# B&R Automation Studio project Doctor
Automation Studio 4.9

## Configuration 5Drive

CPU 4PPC70.0702-20B, AutomationRuntime J4.93, Build 4.1.2, Vc V4.72.6

### Hardware
```
4PPC70_0702_20B : 4PPC70.0702-20B v1.5.4.0
  Connector IF2:
    ActivateDevice = 1
  ConfigurationID = TensionCtl_Config1
  FileDevice1
  FileDeviceName1 = USER
  FileDevicePath1 = USER_PATH
  KeyMappingFile = VC\4PPC70_0702_20B.dis
```

## Configuration Doctoring

CPU 4PPC70.0702-20B, AutomationRuntime J4.93, Build 4.1.2, Safety 0.0, Vc V4.73.3

### Task classes (Cpu.sw)
```
Cyclic#1 (cycle 2000 us, tolerance 4000 us):
  HS_Inp_Doc <- Doctoring.HS_Inp_Doct.prg
  EPLCom_Drv <- EPLCom.EPLCom_Drv1.prg
Cyclic#2 (cycle 10000 us):
  LS_Inp_OP <- Doctoring.LS_Inp_OP.prg
Cyclic#4:
  HMI <- HMI.prg
  Alarms <- Alarms.prg
  EPLCom_Dr1 <- EPLCom.EPLCom_Drv2.prg
DataObjects: Acp10sys
VcDataObjects: Vis <- Vis.dob
Binaries: udbdef, FWRules, TCData, vcctext, arialbd, vcpdi855, vcmgr, vcdsint, vcdsloc, vcbclass, vcfntttf, vctcal, vcshared, vcrt, vcpk, vccbmp, vcfile, vccbtn, vccslider, vccdt, vcptelo, vcalarm, vccnum, vcpdsw, arial, vccovl, vccalarm, vccstr, vcpdi815, vcpfppc7, vcgclass, vcpdihd, vcnet, Vis01, Vis03, vcpkat, Vis02, vcpdvnc, vccline, visvc, vclibvc, vcclbox, vccshape, acp10cfg, Acp10map, arconfig, User, iomap, asfw, ashwac, ashwd, sysconf, Role, vcpfar00, vcxml, vcchspot, vcchtml, vccurl, Vis_Re02, Vis_Re01, Vis_Re03, Vis_Re, vcctrend
Libraries: NcGlobal, sys_lib, brsystem, runtime, LoopConR, LoopCont, Acp10_MC, Acp10man, Acp10par, AsBrMath, Acp10sim, asstring, standard, vclib, visapi, AsEPL, Library, astime, fileio, powerlnk, asieccon, dataobj, vcresman
```

### Hardware
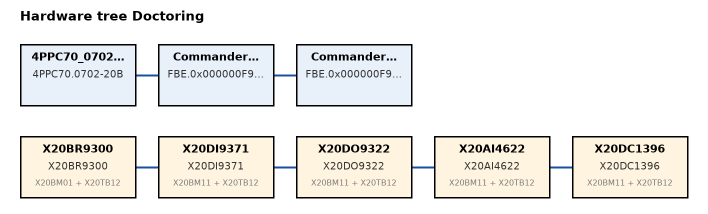
```
4PPC70_0702_20B : 4PPC70.0702-20B v1.5.4.0
  Connector IF1:
    CycleTime = 500
    MuxPrescaler = 2
  Connector IF2:
    ActivateDevice = 1
    Mode = Manual
    InternetAddress = 192.168.111.50
    SubnetMask = 255.255.255.0
    InaNodeNumber = 3
    Vnc1
    VncVcObjectName1 = Vis
    VncKeyMappingFile1 = VC\PS2-Keyboard.dis
    VncAuthentication1 = 1
    VncPasswordViewControl1 = v
    ActivateSnmp = 2
  Connector IF5:
    CycleTime = 1000
    BusLength = 500
  ConfigurationID = TensionCtl_Config1
  SimulationInaNodeNumber = 3
  PermanentPvSize = 5000
  RemanentGlobalPvSize = 10000
  EnableUsbRemoteInstall = 1
  EnableCfRemoteInstall = 1
  RebootReset = 2
  Connections = 8
  TimerDeviceType = EPLX2X
  TimerDevice = 4PPC70_0702_20B.IF1
  IdleTaskClass = 4
  TaskClassIdleTime = 4000
  Cyclic1Duration = 2000
  Cyclic1Tolerance = 4000
  Cyclic2Duration = 10000
  Cyclic5Duration = 500000
  Cyclic5Tolerance = 500000
  FileDevice1
  FileDeviceName1 = USER
  FileDevicePath1 = USER_PATH
  ActivateOpcUa = 1
  OpcUaInformationModels_PV_Version = 1
  VcObjectName = Vis
  KeyMappingFile = VC\4PPC70_0702_20B.dis
Commander_C200_RFC_UnWind : FBE.0x000000F9_Commander C200 RFC_A vV01.01.12.04 (OrderNumber=Commander C200 RFC_A)  [PLK1 -> 4PPC70_0702_20B.IF1 (NodeNumber=3) [Cable Type=PowerlinkCable, Length=10, Version=1.0.0.3]; PLK2 -> Commander_C200_RFC_Wind.PLK1 (NodeNumber=3) [Cable Type=PowerlinkCable, Length=10, Version=1.0.0.3]]
  DummyDeviceType = on
  p2001s05_direction = wo
  p2001s05_value = 5
  p2001s15_value = 0
  p2001s18_direction = wo
  p2004s01_direction = ro
  p2005s01_direction = ro
  p2005s03_direction = ro
  p2005s04_direction = ro
  p2007s01_direction = ro
  p200Es08_value = 0
  p200Es19_value = 0
  p2014s15_value = 
  p6040_value = 0
Commander_C200_RFC_Wind : FBE.0x000000F9_Commander C200 RFC_A vV01.01.12.04 (OrderNumber=Commander C200 RFC_A)  [PLK1 -> Commander_C200_RFC_UnWind.PLK2 (NodeNumber=4) [Cable Type=PowerlinkCable, Length=10, Version=1.0.0.3]]
  p2001s05_direction = wo
  p2001s18_direction = wo
  p2004s01_direction = ro
  p2005s01_direction = ro
  p2005s03_direction = ro
  p2005s04_direction = ro
X20AI4622 : X20AI4622 v1.5.0.0  [SS1 -> X20TB12g.SS; SL -> X20BM11f.SL1]
  Supervision = off
X20BM01 : X20BM01 v2.2.0.0
X20BM11b : X20BM11 v1.1.0.0  [X2X1 -> X20BM01.X2X2]
X20BM11d : X20BM11 v1.1.0.0  [X2X1 -> X20BM11b.X2X2]
X20BM11f : X20BM11 v1.1.0.0  [X2X1 -> X20BM11d.X2X2]
X20BM11h : X20BM11 v1.1.0.0  [X2X1 -> X20BM11f.X2X2]
X20BR9300 : X20BR9300 v1.3.0.0  [SS1 -> X20TB12.SS; SL -> X20BM01.SL1; X2X1 -> 4PPC70_0702_20B.IF5 [Cable Type=X2XCable, Length=10, Version=1.0.0.3]]
  Supervision = off
X20DC1396 : X20DC1396 v1.4.0.0  [SS1 -> X20TB12i.SS; SL -> X20BM11h.SL1]
  Supervision = off
X20DI9371 : X20DI9371 v1.6.0.0  [SS1 -> X20TB12c.SS; SL -> X20BM11b.SL1]
  Supervision = off
X20DO9322 : X20DO9322 v1.6.0.0  [SS1 -> X20TB12e.SS; SL -> X20BM11d.SL1]
  Supervision = off
  StatusInfo = off
X20TB12 : X20TB12 v1.0.0.0
X20TB12c : X20TB12 v1.0.0.0
X20TB12e : X20TB12 v1.0.0.0
X20TB12g : X20TB12 v1.0.0.0
X20TB12i : X20TB12 v1.0.0.0
```

### Cpu.per - 4PPC70_0702_20B/Cpu.per
```iecst
VAR_CONFIG
	Wind AT %M0; (* *)
	UnWind AT %M220; (* *)
	Idler AT %M440; (* *)
END_VAR
```

### IoMap.iom - 4PPC70_0702_20B/IoMap.iom
```iecst
VAR_CONFIG
	Cyclic#1.::AI1[0] AT %IW."X20AI4622".AnalogInput01;
	Cyclic#1.::AI1[1] AT %IW."X20AI4622".AnalogInput02;
	Cyclic#1.::AI1[2] AT %IW."X20AI4622".AnalogInput03;
	Cyclic#1.::AI1[3] AT %IW."X20AI4622".AnalogInput04;
	::Enc_Value AT %IW."X20DC1396".Encoder01;
	::Drive_RW[0].Read_INT[0] AT %IW."Commander_C200_RFC_UnWind".Parameter40_StatusWord_I200A_S28;
	::Drive_RW[0].Write_UINT[0] AT %QW."Commander_C200_RFC_UnWind".Parameter5_JogReference_I2001_S05Out;
	Cyclic#2.::DI1[0] AT %IX."X20DI9371".DigitalInput01;
	Cyclic#2.::DI1[1] AT %IX."X20DI9371".DigitalInput02;
	Cyclic#2.::DI1[2] AT %IX."X20DI9371".DigitalInput03;
	Cyclic#2.::DI1[3] AT %IX."X20DI9371".DigitalInput04;
	Cyclic#2.::DI1[4] AT %IX."X20DI9371".DigitalInput05;
	Cyclic#2.::DI1[5] AT %IX."X20DI9371".DigitalInput06;
	Cyclic#2.::DI1[6] AT %IX."X20DI9371".DigitalInput07;
	Cyclic#2.::DI1[7] AT %IX."X20DI9371".DigitalInput08;
	Cyclic#2.::DI1[8] AT %IX."X20DI9371".DigitalInput09;
	Cyclic#2.::DI1[9] AT %IX."X20DI9371".DigitalInput10;
	Cyclic#2.::DI1[10] AT %IX."X20DI9371".DigitalInput11;
	Cyclic#2.::DI1[11] AT %IX."X20DI9371".DigitalInput12;
	Cyclic#2.::DO1[0] AT %QX."X20DO9322".DigitalOutput01;
	Cyclic#2.::DO1[1] AT %QX."X20DO9322".DigitalOutput02;
	Cyclic#2.::DO1[2] AT %QX."X20DO9322".DigitalOutput03;
	Cyclic#2.::DO1[3] AT %QX."X20DO9322".DigitalOutput04;
	Cyclic#2.::DO1[4] AT %QX."X20DO9322".DigitalOutput05;
	Cyclic#2.::DO1[5] AT %QX."X20DO9322".DigitalOutput06;
	Cyclic#2.::DO1[6] AT %QX."X20DO9322".DigitalOutput07;
	Cyclic#2.::DO1[7] AT %QX."X20DO9322".DigitalOutput08;
	Cyclic#2.::DO1[8] AT %QX."X20DO9322".DigitalOutput09;
	Cyclic#2.::DO1[9] AT %QX."X20DO9322".DigitalOutput10;
	Cyclic#2.::DO1[10] AT %QX."X20DO9322".DigitalOutput11;
	Cyclic#2.::DO1[11] AT %QX."X20DO9322".DigitalOutput12;
	::Drive_RW[0].Read_DINT[1] AT %ID."Commander_C200_RFC_UnWind".Parameter69_ReferenceInRpm_I2001_S45;
	::Drive_RW[0].Read_DINT[2] AT %ID."Commander_C200_RFC_UnWind".Parameter1_OutputFrequency_I2005_S01;
	::Drive_RW[0].Write_UINT[1] AT %QW."Commander_C200_RFC_UnWind".ControlWord_U16_I6040;
	::Drive_RW[0].Read_DINT[0] AT %ID."Commander_C200_RFC_UnWind".Parameter1_CurrentMagnitude_I2004_S01;
	::Drive_RW[0].Read_DINT[1] AT %ID."Commander_C200_RFC_UnWind".Parameter4_MotorRpm_I2005_S04;
	::Drive_RW[0].Read_DINT[3] AT %ID."Commander_C200_RFC_UnWind".Parameter3_OutputPower_I2005_S03;
	::Drive_RW[0].Write_DINT[0] AT %QD."Commander_C200_RFC_UnWind".Parameter22_PresetReference2_I2001_S16Out;
	::Drive_RW[1].Write_UINT[0] AT %QW."Commander_C200_RFC_Wind".Parameter5_JogReference_I2001_S05Out;
	::Drive_RW[1].Write_DINT[0] AT %QD."Commander_C200_RFC_Wind".Parameter22_PresetReference2_I2001_S16Out;
	::Drive_RW[1].Read_DINT[0] AT %ID."Commander_C200_RFC_Wind".Parameter1_CurrentMagnitude_I2004_S01;
	::Drive_RW[1].Read_DINT[2] AT %ID."Commander_C200_RFC_Wind".Parameter1_OutputFrequency_I2005_S01;
	::Drive_RW[1].Read_DINT[3] AT %ID."Commander_C200_RFC_Wind".Parameter3_OutputPower_I2005_S03;
	::Drive_RW[1].Read_DINT[1] AT %ID."Commander_C200_RFC_Wind".Parameter4_MotorRpm_I2005_S04;
	::Drive_RW[0].Read_INT[0] AT %IW."Commander_C200_RFC_UnWind".Parameter1_AnalogueInput1_I2007_S01;
	::Drive_RW[0].Write_DINT[0] AT %QD."Commander_C200_RFC_UnWind".Parameter21_PresetReference1_I2001_S15Out;
	::Drive_RW[0].Write_DINT[0] AT %QD."Commander_C200_RFC_UnWind".Parameter24_PresetReference4_I2001_S18Out;
	::Drive_RW[1].Write_DINT[0] AT %QD."Commander_C200_RFC_Wind".Parameter24_PresetReference4_I2001_S18Out;
END_VAR
```

## Configuration WndCLTensCtrl

### Acp10map.ncm - X20CP1586/Motion/Acp10map.ncm
```
NcMapping (NcSwId=Acp10, DisabledNodesAreHidden=False)
  NcObject gWinderAx (ModuleId=8V1022.001-2, Type=ncAXIS, Channel=1, AcoposSimulation=Complete, InitParameter=gWinderAxi, AcoposParameter=gWinderAxa, Disabled=FALSE, ModuleDisabled=FALSE)  // simulated winder axis
  NcObject gLineAx (ModuleId=8V1022.001-2, Type=ncV_AXIS, Channel=1, InitParameter=gLineAxi, AcoposParameter=gLineAxa, Disabled=FALSE, ModuleDisabled=FALSE)  // virtual master axis
```

## Configuration WndDcrCtrl

### Hardware
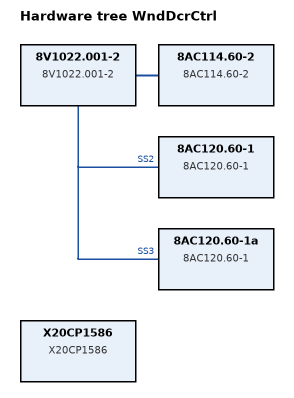
```
8AC114.60-2 : 8AC114.60-2 v1.0.0.8  [SS -> 8V1022.001-2.SS1; PLK1 -> X20CP1586.IF3 (NodeNumber=1) [Cable Type=PowerlinkCable, Length=10, Version=1.0.0.3]]
8AC120.60-1 : 8AC120.60-1 v2.2.0.0  [SS -> 8V1022.001-2.SS2]
8AC120.60-1a : 8AC120.60-1 v2.2.0.0  [SS -> 8V1022.001-2.SS3]
8V1022.001-2 : 8V1022.001-2 v2.2.0.0
  Simulate = complete
  ActiveMotorSimulation_r1 = on
  BothEndSwitchesAreNormallyOpen_r1 = on
  QuickStopIsNormallyOpen_r1 = on
X20CP1586 : X20CP1586 v1.10.0.0
  Connector IF1:
    ActivateIna = 0
  Connector IF2:
    ActivateDevice = 1
    EthInterfaceRedundant = 0
    InaPort = 11160
    Vnc1
    VncVcObjectName1 = Visu
    VncKeyMappingFile1 = VC\PS2-Keyboard.dis
    VncAuthentication1 = 1
    VncPasswordViewOnly1 = v
    VncPasswordViewControl1 = c
  Connector IF3:
    DNAConfiguration = manual
  ConfigurationID = DancerControl_Simulation
  Simulation = 1
  TimerDeviceType = SWIOTIMER
  SystemTick = 400
  TaskClassIdleTime = 400
  Cyclic1Duration = 400
  Cyclic1Tolerance = 0
  Cyclic2Duration = 800
  Cyclic2Tolerance = 0
  Cyclic3Duration = 10000
  Cyclic3Tolerance = 0
  Cyclic4Duration = 100000
  Cyclic4Tolerance = 100000
  Cyclic5Duration = 200000
  Cyclic5Tolerance = 200000
  Cyclic6Duration = 500000
  Cyclic6Tolerance = 500000
  Cyclic7Duration = 1000000
  Cyclic7Tolerance = 1000000
  Cyclic8Duration = 10000
  Cyclic8Tolerance = 30000000
```

### Acp10cfg.ncc - X20CP1586/Motion/Acp10cfg.ncc
```
NcConfiguration (Version=2.48.1, NcSwId=Acp10)
  ACP10CF1_typ:
    cnt_nettrc_rec_drive = 1500
    bufsize_trace_upload = 1200
    tc_nc_man_task = Cyclic #1
    glob_pv_as_ncobject = Yes
    ncsys_dl_broadcast = Yes
    ncsys_dl_acp_reset = Yes
    safemc_log_err_to_ax = Yes
    network_init:
      ncsw_init_execute = Yes
      automatic_execute = No
      node_nr_warning = Yes
      net_err_before_ncact = Yes
    nettrc:
      enter_parsecrec = Yes
      enter_ncaction = Yes
      save_ring_startidx = Yes
    cam_prof_download:
      cam_dat_dl_parallel = No
      tc_cam_dl_parallel = Task class for NC Manager task
    plk_if[0]:
      if_name = SL1.IF2
      tc_CycDat_PLCopen = Task class for NC Manager task
      mc_broadcast_extdat = No
    plk_if[1]:
      if_name = IF3
      tc_CycDat_PLCopen = Task class for NC Manager task
      mc_broadcast_extdat = No
```

### PvMap.vvm - X20CP1586/PvMap.vvm
```iecst
(*Simulation model input parameters*)
VAR_CONFIG
	Cyclic#3.::gControl.Winder.Power AT %Q.::SimModel:SimulationModel.Enable; (*Enable simulation modell if machine is ready*)
	Cyclic#3.::gControl.Line.SetVelocity AT %Q.::SimModel:SetLineVelocity; (*Connect control structure with simulation model*)
	Cyclic#3.::gControl.Winder.SetVelocity AT %Q.::SimModel:SetWinderVelocity; (*Connect control structure with simulation model*)
	Cyclic#3.::gControl.Winder.VelocityCorrection AT %Q.::SimModel:WinderVelocityCorrection; (*Connect control structure with simulation model*)
	Cyclic#3.::gControl.Winder.SetMotorTorque AT %Q.::SimModel:SetMotorTorque; (*Connect control structure with simulation model*)
	Cyclic#3.::gControl.Winder.InitSpeedController AT %Q.::SimModel:InitSpeedController; (*Connect control structure with simulation model*)
	Cyclic#3.::gControl.Winder.ActProportionalGain AT %Q.::SimModel:ActProportionalGain; (*Connect control structure with simulation model*)
	Cyclic#3.::gControl.Winder.ActIntegrationTime AT %Q.::SimModel:ActIntegrationTime; (*Connect control structure with simulation model*)
END_VAR
(*Simulation model output parameters*)
VAR_CONFIG
	::SimModel:SimulationModel.ActLinePosition AT %Q.Cyclic#2.::gControl.Line.ActPosition; (*Connect simulation model with control structure*)
	::SimModel:SimulationModel.ActWinderPosition AT %Q.Cyclic#2.::gControl.Winder.ActPosition; (*Connect simulation model with control structure*)
	::SimModel:SimulationModel.ActDancerPosition AT %Q.Cyclic#2.::gControl.ActDancerPosition; (*Connect simulation model with control structure*)
	::SimModel:SimulationModel.ActLineVelocity AT %Q.Cyclic#2.::gControl.Line.ActVelocity; (*Connect simulation model with control structure*)
	::SimModel:SimulationModel.ActWinderVelocity AT %Q.Cyclic#2.::gControl.Winder.ActVelocity; (*Connect simulation model with control structure*)
	::SimModel:SimulationModel.ActMotorTorque AT %Q.Cyclic#2.::gControl.Winder.ActMotorTorque; (*Connect simulation model with control structure*)
END_VAR
```

## Logical view

Binary libraries used (declarations not repeated): Acp10_MC 3.13.1, vclib

### Global.typ - Global data types
```iecst
TYPE
	ActVal_typ : 	STRUCT
		Input_Val : INT;
		Output_Val : INT;
		Scale : Scale_typ;
	END_STRUCT;
	Ax_GeneralRef : 	STRUCT
		MPM : MPM_Scale;
		RPM : RPM_Scale;
		PulsesPerRev : INT;
		MotorRating : MotorRating_typ;
	END_STRUCT;
	Ax_NonTensionCtl : 	STRUCT
		MPM : MPM_typ;
		Enable : BOOL;
		RPM : RPM_typ;
		Drive : Drive_typ;
		Dia : Diameter_Scale;
		StartingDia : UINT;
		MotorRating : MotorRating_typ;
	END_STRUCT;
	Ax_TensionCtl : 	STRUCT
		Tension : Tension_typ;
		MPM : MPM_typ;
		Enable : BOOL;
		RPM : RPM_typ;
		Drive : Drive_typ;
		Dia : Diameter_Scale;
		StartingDia : UINT;
		MotorRating : MotorRating_typ;
	END_STRUCT;
	Diameter_Scale : 	STRUCT
		InpMPM : INT;
		InpRPM : INT;
		ActDia : INT;
		MinDia : INT;
		MaxDia : INT;
	END_STRUCT;
	DigInp_typ : 	STRUCT
		Emergency_OK : BOOL;
		Jog_mode : BOOL;
		Production_mode : BOOL;
		MPM_Increase : BOOL;
		MPM_Decrease : BOOL;
		Safety_Trip : BOOL;
		Spare1 : BOOL;
		Spare2 : BOOL;
		Spare3 : BOOL;
		Spare4 : BOOL;
		Spare5 : BOOL;
		Spare6 : BOOL;
		Spare7 : BOOL;
		Spare8 : BOOL;
		Spare9 : BOOL;
		Spare10 : BOOL;
	END_STRUCT;
	DigOp_typ : 	STRUCT
		DriveOK : ARRAY[0..6]OF BOOL;
		Production_Enable : BOOL;
		Alarm_Lamp : BOOL;
		Safety_Trip : BOOL;
		Spare1 : BOOL;
		Spare2 : BOOL;
		Spare3 : BOOL;
		Spare4 : BOOL;
		Spare5 : BOOL;
		Spare6 : BOOL;
		Spare7 : BOOL;
		Spare8 : BOOL;
		Spare9 : BOOL;
		Spare10 : BOOL;
	END_STRUCT;
	Drive_typ : 	STRUCT
		Freq_Scal : Scale_typ;
		RPM_Scal : Scale_typ;
		Trq_Scal : Scale_typ;
		Current_Scal : Scale_typ;
		ActFreq : INT;
		Status : USINT;
		ActualTrq : INT;
		ActualAmp : INT;
		ActRPM : INT;
		Fault : USINT;
		Drive_Healthy : BOOL;
		Drive_Enable : BOOL;
	END_STRUCT;
	MPM_Scale : 	STRUCT
		InpDia : INT;
		InpRPM : INT;
		ActMPM : INT;
	END_STRUCT;
	MPM_typ : 	STRUCT
		SetMPM : INT;
		ActualMPM : INT;
		Enable : BOOL;
		Set : SetVal_typ;
		Actual : ActVal_typ;
	END_STRUCT;
	PIDPara_typ : 	STRUCT
		Y_max : INT;
		Y_min : INT;
		dY_max : REAL;
		Kp_sta : REAL;
		Tn_sta : REAL;
		Tv_sta : REAL;
		Tf_sta : REAL;
		WindDamp : REAL;
		Fbk_mode : REAL;
		d_mode : USINT;
		calc_mode : USINT;
		Attenu_val : REAL;
		Update : BOOL;
		Kp_mov : USINT;
		Tn_mov : USINT;
		Tv_mov : USINT;
		Tf_mov : USINT;
	END_STRUCT;
	RPM_Scale : 	STRUCT
		InpMPM : INT;
		InpDia : INT;
		ActRPM : INT;
		InpBits : INT;
	END_STRUCT;
	RPM_typ : 	STRUCT
		SetRPM : INT;
		ActualRPM : INT;
		Enable : BOOL;
		Set : SetVal_typ;
		Actual : ActVal_typ;
		PulsesPerRev : INT;
		GearRatio : USINT;
	END_STRUCT;
	Scale_typ : 	STRUCT
		InMin : INT;
		InMax : INT;
		OutMin : INT;
		OutMax : INT;
		Filter_tim : INT;
	END_STRUCT;
	SetVal_typ : 	STRUCT
		Output_Val : INT;
		Input_Val : INT;
		Scale : Scale_typ;
	END_STRUCT;
	Tension_typ : 	STRUCT
		Actual : ActVal_typ;
		Set : SetVal_typ;
		Enable : BOOL;
		SetTension : INT;
		ActualTension : INT;
		PID : PID_typ;
	END_STRUCT;
	DriveRW_typ : 	STRUCT
		Read_BOOL : ARRAY[0..9]OF BOOL;
		Read_UINT : ARRAY[0..9]OF UINT;
		Read_INT : ARRAY[0..9]OF INT;
		Read_USINT : ARRAY[0..9]OF USINT;
		Read_DINT : ARRAY[0..9]OF DINT;
		Read_UDINT : ARRAY[0..9]OF UDINT;
		Write_BOOL : ARRAY[0..9]OF BOOL;
		Write_INT : ARRAY[0..9]OF INT;
		Write_UINT : ARRAY[0..9]OF UINT;
		Write_USINT : ARRAY[0..9]OF USINT;
		Write_DINT : ARRAY[0..9]OF DINT;
		Write_UDINT : ARRAY[0..9]OF UDINT;
	END_STRUCT;
	MotorRating_typ : 	STRUCT
		RatedFreq : DINT;
		RatedCurrent : DINT;
		RatedSpeed : DINT;
		RatedVoltage : INT;
		RatedPF : INT;
	END_STRUCT;
	PID_typ : 	STRUCT
		Prop_Gain : INT;
		Intg_Gain : INT;
		Derv_Gain : INT;
		UpperLimit : INT;
		LowerLimit : INT;
		Enable : USINT;
		Reference_Add : INT;
		Feedback_Add : INT;
		Output : INT;
		Error : INT;
	END_STRUCT;
END_TYPE
```

### Global.var - Global variables
```iecst
VAR
	AI1 : ARRAY[0..4] OF INT;
	AI2 : ARRAY[0..3] OF INT;
	AI3 : ARRAY[0..4] OF INT;
	Alarm : ARRAY[0..99] OF BOOL;
	Alarm_cnt : USINT;
	Alarm_mc : ARRAY[0..99] OF BOOL;
	Alarm_new : BOOL;
	AO1 : ARRAY[0..3] OF INT;
	Axis_Motor : INT;
	Backbtn : INT;
	CurrPage : USINT;
	DataRead_INT : {REDUND_UNREPLICABLE} INT := 0;
	DataRead_UINT : UINT;
	DataTobeRead_INT : INT;
	DataTobeSent_UINT : UINT;
	DI1 : ARRAY[0..11] OF BOOL;
	DI2 : ARRAY[0..11] OF BOOL;
	DigInp : DigInp_typ;
	DigOp : DigOp_typ;
	DO1 : ARRAY[0..11] OF BOOL;
	DO2 : ARRAY[0..11] OF BOOL;
	Drive_RW : ARRAY[0..4] OF DriveRW_typ;
	DrvComm : BOOL;
	Enc_Value : INT;
	error : UINT;
END_VAR
VAR RETAIN
	Idler : Ax_GeneralRef;
END_VAR
VAR
	InFeed : Ax_TensionCtl;
END_VAR
VAR CONSTANT
	INFEED : USINT := 1;
END_VAR
VAR
	LastPage : USINT;
	LoginSuccessful : BOOL;
END_VAR
VAR CONSTANT
	MAIN : USINT := 4;
END_VAR
VAR
	MainDrive : Ax_NonTensionCtl;
END_VAR
VAR CONSTANT
	MAX_AXES : USINT := 5;
END_VAR
VAR
	NewPage : USINT;
	NewPageReq : USINT;
	OutFeed : Ax_TensionCtl;
END_VAR
VAR CONSTANT
	OUTFEED : USINT := 2;
END_VAR
VAR
	PageCall : BOOL;
	ParamChange : BOOL;
END_VAR
VAR CONSTANT
	PLC_INTF : STRING[20] := 'IF1';
END_VAR
VAR
	PrevPage : USINT;
	PrevPageTemp : USINT;
END_VAR
VAR CONSTANT
	PulsesPerRev : INT := 0;
END_VAR
VAR
	PulsesPerSec : INT;
	SavePID : BOOL;
	Save : BOOL;
	Statusdp_alarm : UINT;
	Statusdp_blink : UINT;
	status_gettime : UINT;
	TempPropGain : INT;
	TempIntgGain : INT;
	TempDervGain : INT;
	TempPIDFeedback : INT;
	TempPIDRef : INT;
	TempCurrent : DINT;
	TempFreq : DINT;
	TempPF : INT;
	TempSpeed : DINT;
	TempVoltage : INT;
END_VAR
VAR RETAIN
	UnWind : Ax_TensionCtl;
END_VAR
VAR CONSTANT
	UNWINDER : USINT := 0;
END_VAR
VAR
	UnWindpara : LCPIDpara;
	UserAccessLevel : USINT;
END_VAR
VAR RETAIN
	Wind : Ax_TensionCtl;
END_VAR
VAR CONSTANT
	WINDER : USINT := 3;
END_VAR
VAR
	Tune_Enable : BOOL;
	Axis_MotorTune : USINT;
END_VAR
```


### Program Logical/UnWindTC (IEC)

#### Cyclic.st
```iecst
PROGRAM _CYCLIC
	(* Insert code here *)
	(* PID parameters *)
	LCPIDpara_0.enable := start;
	LCPIDpara_0.enter  := paraEnter;
	LCPIDpara_0();		(* LCPIDpara function block call *)
	paraEnter := 0;

	(* PID controller *)
	LCPID_0.enable   := start;
	LCPID_0.ident    := LCPIDpara_0.ident; (* ident of PIDpara -> provides parameters (Kp, Tn, Tv, ...) *)
	LCPID_0.W        := setValue;
	LCPID_0.X        := actValue;
	LCPID_0.basetime := baseLCCounter.mscnt;
	LCPID_0();		(* LCPID function block call *)
	manipulatedVar := LCPID_0.Y;

END_PROGRAM
```

#### Init.st
```iecst
PROGRAM _INIT
	(* Insert code here *)
	(* Parameters for PID controller *)
	UnWindPID.A        := 0;
	UnWindPID.Y_man    := 0;
	UnWindPID.Y_fbk    := 0;
	UnWindPID.hold_I   := FALSE;
	UnWindPID.out_mode := LCPID_OUT_MODE_AUTO;

	(* Parameters for PID controller *)
	LCPID_0.A        := 0;
	LCPID_0.Y_man    := 0;
	LCPID_0.Y_fbk    := 0;
	LCPID_0.hold_I   := FALSE;
	LCPID_0.out_mode := LCPID_OUT_MODE_AUTO;

	(* Parameters for PT2 element *)
	LCRPT2_0.V     := 0.039;
	LCRPT2_0.T1    := 0.9;
	LCRPT2_0.T2    := 15.3;
	LCRPT2_0.y_set := 0.0;
	LCRPT2_0.set   := 0;

END_PROGRAM
```

### Program Logical/HMI (IEC)

#### Variables.var
```iecst
VAR
	CheckCredentials : BOOL;
	ErrorMessage : STRING[80];
	i : INT;
	Init : BOOL;
	InputPassword : STRING[80]; (*Input taken from HMI*)
	InputUsername : STRING[80]; (*Input taken from HMI*)
	CurrentYear : UINT;
	CurrentSecond : USINT;
	CurrentMonth : USINT;
	CurrentMinute : USINT;
	CurrentHour : USINT;
	CurrentDay : USINT;
	NewYear : UINT;
	NewSecond : USINT;
	NewMonth : USINT;
	NewMinute : USINT;
	NewHour : USINT;
	NewDay : USINT;
	DateTimeSet : UINT; (*Confirms if new date/time was set successfully*)
	SetNewDateTime : BOOL; (*Trigger to apply new date/time*)
	RTC_Get : RTCtime_typ; (*Structure to read current date and time*)
	RTC_Set : RTCtime_typ; (*Structure to set current date and time*)
	Status_RTC : UINT;
	temp_var : BOOL;
	startdly : BOOL;
	dlycnt : USINT;
	WelcomeTimer : TON_10ms;
END_VAR
```

#### Cyclic.st
```iecst
PROGRAM _CYCLIC
	// Time
	// Reads current date/time from PLC's RTC

	RTC_gettime(ADR(RTC_Get));  // Call PLC's built-in RTC function

	// Update outputs for display
	CurrentYear   := RTC_Get.year;
	CurrentMonth  := RTC_Get.month;
	CurrentDay    := RTC_Get.day;
	CurrentHour   := RTC_Get.hour;
	CurrentMinute := RTC_Get.minute;
	CurrentSecond := RTC_Get.second;

	// Set Date and Time when 'Set Date Time' button is pressed
	IF SetNewDateTime THEN
		IF(temp_var = 0)THEN
			Status_RTC	:= 1;
			temp_var	:= 1;
		END_IF

		RTC_Set.year    := NewYear;
		RTC_Set.month   := NewMonth;
		RTC_Set.day     := NewDay;
		RTC_Set.hour    := NewHour;
		RTC_Set.minute  := NewMinute;
		RTC_Set.second  := NewSecond;

		// Call RTC set function
		Status_RTC := RTC_settime(ADR(RTC_Set));  // Returns TRUE if successful

		IF(Status_RTC = 0)THEN
			SetNewDateTime	:= 0;
			temp_var		:= 0;
		END_IF

	END_IF;

	// Login check
	//IF(CurrPage > 0 AND CurrPage < 13) THEN
	IF (InputUsername = 'Admin' AND InputPassword = '1234') THEN
		LoginSuccessful := TRUE;
		UserAccessLevel := 1;	// Full access
		CheckCredentials := TRUE;
		ErrorMessage := 'Logged in';
	ELSE
		LoginSuccessful := FALSE;
		UserAccessLevel := 0;	// No input access
		CheckCredentials := FALSE;
		ErrorMessage := 'Wrong user name or password';
	END_IF;

	ErrorMessage := '';   	// Clear any previous message
	InputUsername := '';	// Clear InputUsername field
	InputPassword := '';	// Clear InputPassword field
	//END_IF

	IF(Alarm_new = 1)THEN
		Statusdp_alarm	:= 0;
	ELSE
		Statusdp_alarm	:= 1;
	END_IF

	IF((NewPageReq <> CurrPage) AND (dlycnt = 0)) THEN
		PrevPage := CurrPage;
		NewPage := NewPageReq;
		startdly	:= 0;
	END_IF

	IF(Backbtn = 1) THEN
		PrevPageTemp 	:= PrevPage;
		PrevPage 		:= CurrPage;
		NewPage 		:= PrevPageTemp;
		startdly		:= 1;
		Backbtn 		:= 0;
	END_IF

	IF((CurrPage = 0)AND (NewPageReq = 0))THEN
		WelcomeTimer.IN	:= 1;
		WelcomeTimer.PT	:= 500;
		IF(WelcomeTimer.Q = 1)THEN
			NewPageReq		:= 1;
			WelcomeTimer.IN	:= 0;
		END_IF
	END_IF

	WelcomeTimer();

	IF(startdly = 1)THEN
		dlycnt 		:= dlycnt + 1;
		NewPageReq 	:= CurrPage;
		IF(dlycnt = 3)THEN
			startdly	:= 0;
			dlycnt		:= 0;
		END_IF
	END_IF

END_PROGRAM
```

#### Init.st
```iecst
PROGRAM _INIT
		(*Input of Tension Sensor for 4 axes except main drive *)
	AI1[0]	:= 0;	(*Unwinder Loadcell *)
	AI1[1]	:= 0;	(* Infeed Loadcell *)
	AI1[2]	:= 0;	(* Outfeed Loadcell *)
	AI1[3]	:= 0;	(* Winder Load cell *)
	AI1[4]	:= 0;	(* Dummy Load cell for Main Drive *)

	AI2[0]	:= 0;
	AI2[1]	:= 0;
	AI2[2]	:= 0;
	AI2[3]	:= 0; (*This input is configured for MAIN RPM calculation *)

	(* Input for RPM measurement from drive AI for 4 axes except Winder RPM*)
	AI3[0]	:= 0;   (* Unwinder RPM *)
	AI3[1]	:= 0;	(* Infeed RPM *)
	AI3[2]	:= 0;	(* Outfeed RPM *)
	AI3[3]	:= 0;	(* Winder RPM *)
	AI3[4]	:= 0;	(*This input is configured from AI2[3] for MAIN RPM *)

	AO1[0]	:= 0;
	AO1[1]	:= 0;
	AO1[2]	:= 0;
	AO1[3]	:= 0;

	DI1[0]	:= 0;
	DI1[1]	:= 0;
	DI1[2]	:= 0;
	DI1[3]	:= 0;
	DI1[4]	:= 0;
	DI1[5]	:= 0;
	DI1[6]	:= 0;
	DI1[7]	:= 0;
	DI1[8]	:= 0;
	DI1[9]	:= 0;
	DI1[10]	:= 0;
	DI1[11]	:= 0;

	DI2[0]	:= 0;
	DI2[1]	:= 0;
	DI2[2]	:= 0;
	DI2[3]	:= 0;
	DI2[4]	:= 0;
	DI2[5]	:= 0;
	DI2[6]	:= 0;
	DI2[7]	:= 0;
	DI2[8]	:= 0;
	DI2[9]	:= 0;
	DI2[10]	:= 0;
	DI2[11]	:= 0;

	DO1[0]	:= 0;
	DO1[1]	:= 0;
	DO1[2]	:= 0;
	DO1[3]	:= 0;
	DO1[4]	:= 0;
	DO1[5]	:= 0;
	DO1[6]	:= 0;
	DO1[7]	:= 0;
	DO1[8]	:= 0;
	DO1[9]	:= 0;
	DO1[10]	:= 0;
	DO1[11]	:= 0;

	DO2[0]	:= 0;
	DO2[1]	:= 0;
	DO2[2]	:= 0;
	DO2[3]	:= 0;
	DO2[4]	:= 0;
	DO2[5]	:= 0;
	DO2[6]	:= 0;
	DO2[7]	:= 0;
	DO2[8]	:= 0;
	DO2[9]	:= 0;
	DO2[10]	:= 0;
	DO2[11]	:= 0;

	PageCall	:= 0;
	LastPage	:= 0;
	NewPageReq	:= 0;
	PrevPage	:= 0;
	CurrPage	:= 0;
	DrvComm		:= 0;
	Init		:= 1;
	ParamChange	:= 0;
	NewPage		:= 0;
	SetNewDateTime	:= 0;
	Backbtn := 0;
END_PROGRAM
```

### Program Logical/EPLCom/UnWind_Com (IEC)

#### Variables.var
```iecst
VAR
	cnt_enable : BOOL;
	Control_Enable : SINT;
	Control_Enb : USINT;
	Control_WORD : INT;
	DIO_Conf : INT;
	dlycnt : USINT := 0;
	dlycnt1 : USINT;
	dlycnt_pid : USINT;
	dlycnt_wrpid : USINT;
	Drv_Status : INT;
	Ingr_Gain : INT;
	init : INT;
	IntGain_Set : INT;
	NMT_Stat : UDINT;
	Obj_Ident : UDINT;
	rd_step : USINT;
	SDORead1 : EplSDORead;
	SDOWrite : EplSDOWrite;
	SDO_rd : USINT;
	SDO_rd2 : USINT;
	SDO_wr : USINT;
	Status_WORD : INT;
	step : USINT;
	tempstat : UINT;
	tempstat_2 : UINT;
	wrpid_step : USINT;
	wr_step : USINT;
	execonce_rd : BOOL;
	execonce_wr : BOOL;
	SDO_rdinit : BOOL;
	Statuschk_dly : USINT;
	statechg : BOOL;
END_VAR
```

#### Cyclic.st
```iecst
PROGRAM _CYCLIC

	(* Read the Status Word & Control Enable Status on Power ON *)

	IF(SDO_rdinit = 1)THEN
		SDORead1.pData 		:= ADR(Status_WORD); //Data to be read into here
		SDORead1.datalen	:= 2; //Data length, 2 bytes for 16-bit parameter
		SDORead1.index 		:= 16#200A;
		SDORead1.subindex	:= 40;
		SDORead1.enable		:= 1;
		dlycnt				:= dlycnt + 1;
		IF(dlycnt > 1)THEN
			IF (SDORead1.status = 0) THEN
				SDORead1.enable	:= 0;
				dlycnt			:= 0;
				Drv_Status		:= Status_WORD;
			ELSIF(SDORead1.status <> 65535)THEN
				SDORead1.enable	:= 0;
			END_IF
		END_IF

		IF(Drv_Status.0 = 1)THEN
			UnWind.Drive.Drive_Healthy	:= 1;
			Alarm[1]					:= 0;
			SDO_wr						:= 1;	//Update the control word and enable the drive
			Statuschk_dly				:= 0;
			SDO_rdinit					:= 0;
		ELSE
			Statuschk_dly				:= Statuschk_dly + 1;
			IF(Statuschk_dly > 4)THEN
				UnWind.Drive.Drive_Healthy	:= 0;
				Alarm[1]				:= 1;
			END_IF
		END_IF

	END_IF

	(* Initial Power Up Configuring the Control Word to Read Freq. Command from Preset-1 & disable other preset values
	& enable the Control *)

	CASE wr_step OF
		0:
			IF((SDO_wr = 1)AND(init = 1))THEN
				wr_step	:= 1;
				dlycnt1	:= 0;
			END_IF

		1:
			//Disable the Control Enable
			Control_Enable		:= 0;
			SDOWrite.pData		:= ADR(Control_Enable);
			SDOWrite.datalen 	:= 1; //Data length, 2 bytes for 16-bit parameter
			SDOWrite.index 		:= 16#2006;
			SDOWrite.subindex	:= 43;
			SDOWrite.enable		:= 1;
			dlycnt1				:= dlycnt1 + 1;
			IF(dlycnt1 > 1)THEN
				IF (SDOWrite.status = 0) THEN
					SDOWrite.enable	:= 0;
					wr_step			:= 2;
					dlycnt1			:= 0;
				ELSIF(SDOWrite.status <> 65535)THEN
					SDOWrite.enable	:= 0;
					SDO_wr			:= 0;
				END_IF
			END_IF

		2:
			// Set the Control Word to Run at Preset Mode
			Control_WORD		:= 387;	//For preset
			SDOWrite.pData		:= ADR(Control_WORD);
			SDOWrite.datalen 	:= 2; //Data length, 2 bytes for 16-bit parameter
			SDOWrite.index 		:= 16#2006;
			SDOWrite.subindex	:= 42;
			SDOWrite.enable		:= 1;
			dlycnt1				:= dlycnt1 + 1;
			IF(dlycnt1 > 1)THEN
				IF (SDOWrite.status = 0) THEN
					SDOWrite.enable	:= 0;
					wr_step			:= 3;
					dlycnt1			:= 0;
				ELSIF(SDOWrite.status <> 65535)THEN
					SDOWrite.enable	:= 0;
				END_IF
			END_IF
		3:
			DIO_Conf		:= 0;

			SDOWrite.pData		:= ADR(DIO_Conf);
			SDOWrite.datalen 	:= 2; //Data length, 2 bytes for 16-bit parameter
			SDOWrite.index 		:= 16#2008; //Index = 0x2000 + Menu Number
			SDOWrite.subindex	:= 22;
			SDOWrite.enable		:= 1;
			dlycnt1				:= dlycnt1 + 1;
			IF(dlycnt1 > 1)THEN
				IF (SDOWrite.status = 0) THEN
					SDOWrite.enable	:= 0;
					wr_step			:= 4;
					dlycnt1			:= 0;
					//				ELSIF((SDOWrite.status <> 65535)AND(SDOWrite.status <> 65534))THEN
				ELSIF(SDOWrite.status <> 65535)THEN
					SDOWrite.enable	:= 0;
					SDO_wr			:= 0;
				END_IF
			END_IF

		4:
			DIO_Conf		:= 0;

			SDOWrite.pData		:= ADR(DIO_Conf);
			SDOWrite.datalen 	:= 2; //Data length, 2 bytes for 16-bit parameter
			SDOWrite.index 		:= 16#2008; //Index = 0x2000 + Menu Number
			SDOWrite.subindex	:= 23;
			SDOWrite.enable		:= 1;
			dlycnt1				:= dlycnt1 + 1;
			IF(dlycnt1 > 1)THEN
				IF (SDOWrite.status = 0) THEN
					SDOWrite.enable	:= 0;
					wr_step			:= 5;
					dlycnt1			:= 0;
					//				ELSIF((SDOWrite.status <> 65535)AND(SDOWrite.status <> 65534))THEN
				ELSIF(SDOWrite.status <> 65535)THEN
					SDOWrite.enable	:= 0;
					SDO_wr			:= 0;
				END_IF
			END_IF

		5:
			DIO_Conf		:= 0;

			SDOWrite.pData		:= ADR(DIO_Conf);
			SDOWrite.datalen 	:= 2; //Data length, 2 bytes for 16-bit parameter
			SDOWrite.index 		:= 16#2008; //Index = 0x2000 + Menu Number
			SDOWrite.subindex	:= 24;
			SDOWrite.enable		:= 1;
			dlycnt1				:= dlycnt1 + 1;
			IF(dlycnt1 > 1)THEN
				IF (SDOWrite.status = 0) THEN
					SDOWrite.enable	:= 0;
					wr_step			:= 6;
					dlycnt1			:= 0;
				ELSIF(SDOWrite.status <> 65535)THEN
					SDOWrite.enable	:= 0;
					SDO_wr			:= 0;
				END_IF
			END_IF

		6:
			//Enable the Control Word once configured

			Control_Enable		:= 1;
			SDOWrite.pData		:= ADR(Control_Enable);
			SDOWrite.datalen 	:= 1; //Data length, 2 bytes for 16-bit parameter
			SDOWrite.index 		:= 16#2006;
			SDOWrite.subindex	:= 43;
			SDOWrite.enable		:= 1;
			dlycnt1				:= dlycnt1 + 1;
			IF(dlycnt1 > 1)THEN
				IF (SDOWrite.status = 0) THEN
					SDOWrite.enable	:= 0;
					wr_step			:= 0;
					dlycnt1			:= 0;
					SDO_wr			:= 0;
					init			:= 0;
					SDO_rd			:= 1;
					execonce_wr		:= 1;
				ELSIF(SDOWrite.status <> 65535)THEN
					SDOWrite.enable	:= 0;
					SDO_wr			:= 0;
				END_IF
			END_IF

	END_CASE

	(* Once the Control word is configured on Power ON, read the status of the drive *)
	(* Reconfirm that the drives are in Run Mode & Control is enabled *)

	CASE rd_step OF
		0:
			IF((SDO_rd = 1)AND(DO1[0] = 1))THEN
				rd_step		:= 1;
				dlycnt		:= 0;
				Drv_Status	:= 0;
			END_IF
		1:
			// Reconfirm if Status Word still shows drive as Healty

			SDORead1.pData := ADR(Status_WORD); //Data to be read into here
			SDORead1.datalen := 2; //Data length, 2 bytes for 16-bit parameter
			SDORead1.index 		:= 16#200A;
			SDORead1.subindex	:= 40;
			SDORead1.enable		:= 1;
			dlycnt				:= dlycnt + 1;
			IF(dlycnt > 1)THEN
				IF (SDORead1.status = 0) THEN
					SDORead1.enable				:= 0;
					rd_step						:= 2;
					dlycnt						:= 0;
					Drv_Status					:= Status_WORD;
					UnWind.Drive.Drive_Enable	:= Status_WORD.1;

				ELSIF(SDORead1.status <> 65535)THEN
					SDORead1.enable	:= 0;
				END_IF
			END_IF

		2:
			// Reconfirm if Control Word Enable is still 1

			SDORead1.pData 		:= ADR(Status_WORD); //Data to be read into here
			SDORead1.datalen 	:= 1; //Data length, 2 bytes for 16-bit parameter
			SDORead1.index 		:= 16#2006;
			SDORead1.subindex	:= 43;
			SDORead1.enable		:= 1;
			dlycnt				:= dlycnt + 1;
			IF(dlycnt > 1)THEN
				IF (SDORead1.status = 0) THEN
					SDORead1.enable	:= 0;
					rd_step			:= 0;
					dlycnt			:= 0;
					SDO_rd			:= 0;
					execonce_rd		:= 1;
					Control_Enb		:=	INT_TO_USINT(Status_WORD);
				ELSIF(SDORead1.status <> 65535)THEN
					SDORead1.enable	:= 0;
				END_IF
			END_IF
	END_CASE

	(* Disbale SDO read/write once the configuration is done *)
	IF((SDO_rd = 0)AND(execonce_rd = 1))THEN
		SDORead1.enable	:= 0;
		rd_step			:= 0;
		dlycnt			:= 0;
		execonce_rd		:= 0;
	END_IF

	IF((SDO_wr = 0)AND(init = 0)AND(execonce_wr = 1))THEN
		SDOWrite.enable	:= 0;
		wr_step			:= 0;
		dlycnt1			:= 0;
		execonce_wr		:= 0;
	END_IF

	(* AFter Power On, if the SDO Write is triggered then it is to Enable/Disable the drive.
	This enable/Disable is done by forcing the Control_Enable Bit *)

	IF((SDO_wr = 1)AND(init = 0))THEN
		//Control_Enable	:= 0;
		SDOWrite.pData		:= ADR(Control_Enable);
		SDOWrite.datalen 	:= 1; //Data length, 2 bytes for 16-bit parameter
		SDOWrite.index 		:= 16#2006;
		SDOWrite.subindex	:= 43;
		SDOWrite.enable		:= 1;
		dlycnt1				:= dlycnt1 + 1;
		IF(dlycnt1 > 1)THEN
			IF (SDOWrite.status = 0) THEN
				SDOWrite.enable	:= 0;
				wr_step			:= 0;
				dlycnt1			:= 0;
				SDO_wr			:= 0;
				SDO_rd			:= 1;
			ELSIF(SDOWrite.status <> 65535)THEN
				SDOWrite.enable	:= 0;
				SDO_wr			:= 0;
			END_IF
		END_IF
	END_IF

	IF((DigInp.Production_mode = 0)AND(DigInp.Jog_mode = 0)AND(statechg = 1))THEN
		Control_Enable	:= 0;
		SDO_wr			:= 1;
		statechg		:= 0;
	ELSIF((DigInp.Production_mode = 1)OR(DigInp.Jog_mode = 1)AND(statechg = 0))THEN
		statechg		:= 1;
		Control_Enable	:= 1;
		SDO_wr			:= 1;
	END_IF

	SDORead1();
	SDOWrite();

END_PROGRAM
```

#### Init.st
```iecst
PROGRAM _INIT
	(* Insert code here *)
	(* Get NMT Status *)
	SDORead1.enable	:= 0;
	SDORead1.pDevice := ADR(PLC_INTF); //POWERLINK interface on MN (PLC) ‘IF1’
	SDORead1.node := 3; //Node address is set to 3

	SDOWrite.enable		:= 0;
	SDOWrite.node		:= 3;
	SDOWrite.pDevice	:= ADR(PLC_INTF);
	SDOWrite.pData		:= ADR(Control_WORD);

	cnt_enable		:= 0;
	SDO_rdinit		:= 1;
	SDO_rd			:= 0;
	execonce_rd		:= 1;
	init			:= 1;
	SDO_wr			:= 0;
	execonce_wr		:= 0;
	dlycnt			:= 0;
	dlycnt1			:= 0;

END_PROGRAM
```

### Program Logical/EPLCom/Wind_Com (IEC)

#### Variables.var
```iecst
VAR
	cnt_enable : BOOL := 00;
	Control_Enable : INT;
	Control_Enb : USINT := 0;
	Control_WORD : INT;
	DataReceived : UINT;
	DataReceived_INT : INT := 0;
	DerGain_Set : INT;
	Derv_Gain : INT;
	DIO_Conf : INT := 0;
	dlycnt : USINT := 0;
	dlycnt1 : USINT := 0;
	dlycnt_pid : USINT := 0;
	dlycnt_wrpid : USINT;
	Drv_Status : INT := 0;
	Ingr_Gain : INT;
	init : INT;
	IntGain_Set : INT;
	PID_RefSrc : UINT;
	PID_WORD : INT;
	Porp_Gain : INT;
	PropGain_Set : INT;
	Prop_Gain : INT;
	rdpid_step : USINT := 0;
	rd_step : USINT;
	RefSrc_Set : UINT;
	RefSrc_WORD : UINT;
	SDORead1 : EplSDORead;
	SDORead_PID : EplSDORead;
	SDOWrite : EplSDOWrite;
	SDO_pid : BOOL := FALSE;
	SDO_pidwr : BOOL;
	SDO_PIDWR : EplSDOWrite;
	SDO_rd : BOOL := FALSE;
	SDO_wr : USINT := 0;
	Status_WORD : INT := 0;
	wrpid_step : USINT;
	wr_step : USINT := 0;
	TempFreq : DINT;
	TempCurrent : DINT;
	TempVoltage : USINT;
	TempSpeed : USINT;
	TempPF : DINT;
	execonce_wr : BOOL;
	execonce_rd : BOOL;
	SDO_rdinit : BOOL;
	Statuschk_dly : USINT;
	statechg : BOOL;
END_VAR
```

#### Cyclic.st
```iecst
PROGRAM _CYCLIC

	(* Read the Status Word & Control Enable Status on Power ON *)

	IF(SDO_rdinit = 1)THEN
		SDORead1.pData 		:= ADR(Status_WORD); //Data to be read into here
		SDORead1.datalen	:= 2; //Data length, 2 bytes for 16-bit parameter
		SDORead1.index 		:= 16#200A;
		SDORead1.subindex	:= 40;
		SDORead1.enable		:= 1;
		dlycnt				:= dlycnt + 1;
		IF(dlycnt > 1)THEN
			IF (SDORead1.status = 0) THEN
				SDORead1.enable	:= 0;
				dlycnt			:= 0;
				Drv_Status		:= Status_WORD;
			ELSIF(SDORead1.status <> 65535)THEN
				SDORead1.enable	:= 0;
			END_IF
		END_IF

		IF(Drv_Status.0 = 1)THEN
			Wind.Drive.Drive_Healthy	:= 1;
			Alarm[2]					:= 0;
			SDO_wr						:= 1;	//Update the control word and enable the drive
			Statuschk_dly				:= 0;
			SDO_rdinit					:= 0;
		ELSE
			Statuschk_dly				:= Statuschk_dly + 1;
			IF(Statuschk_dly > 4)THEN
				Wind.Drive.Drive_Healthy	:= 0;
				Alarm[2]				:= 1;
			END_IF
		END_IF

	END_IF

	(* Initial Power Up Configuring the Control Word to Read Freq. Command from Preset-1 & disable other preset values
	& enable the Control *)

	CASE wr_step OF
		0:
			IF((SDO_wr = 1)AND(init = 1))THEN
				wr_step	:= 1;
				dlycnt1	:= 0;
			END_IF

		1:
			//Disable the Control Enable
			Control_Enable		:= 0;
			SDOWrite.pData		:= ADR(Control_Enable);
			SDOWrite.datalen 	:= 1; //Data length, 2 bytes for 16-bit parameter
			SDOWrite.index 		:= 16#2006;
			SDOWrite.subindex	:= 43;
			SDOWrite.enable		:= 1;
			dlycnt1				:= dlycnt1 + 1;
			IF(dlycnt1 > 1)THEN
				IF (SDOWrite.status = 0) THEN
					SDOWrite.enable	:= 0;
					wr_step			:= 2;
					dlycnt1			:= 0;
				ELSIF(SDOWrite.status <> 65535)THEN
					SDOWrite.enable	:= 0;
					SDO_wr			:= 0;
				END_IF
			END_IF

		2:
			// Set the Control Word to Run at Preset Mode
			Control_WORD		:= 387;	//For preset
			SDOWrite.pData		:= ADR(Control_WORD);
			SDOWrite.datalen 	:= 2; //Data length, 2 bytes for 16-bit parameter
			SDOWrite.index 		:= 16#2006;
			SDOWrite.subindex	:= 42;
			SDOWrite.enable		:= 1;
			dlycnt1				:= dlycnt1 + 1;
			IF(dlycnt1 > 1)THEN
				IF (SDOWrite.status = 0) THEN
					SDOWrite.enable	:= 0;
					wr_step			:= 3;
					dlycnt1			:= 0;
				ELSIF(SDOWrite.status <> 65535)THEN
					SDOWrite.enable	:= 0;
				END_IF
			END_IF
		3:
			DIO_Conf		:= 0;

			SDOWrite.pData		:= ADR(DIO_Conf);
			SDOWrite.datalen 	:= 2; //Data length, 2 bytes for 16-bit parameter
			SDOWrite.index 		:= 16#2008; //Index = 0x2000 + Menu Number
			SDOWrite.subindex	:= 22;
			SDOWrite.enable		:= 1;
			dlycnt1				:= dlycnt1 + 1;
			IF(dlycnt1 > 1)THEN
				IF (SDOWrite.status = 0) THEN
					SDOWrite.enable	:= 0;
					wr_step			:= 4;
					dlycnt1			:= 0;
					//				ELSIF((SDOWrite.status <> 65535)AND(SDOWrite.status <> 65534))THEN
				ELSIF(SDOWrite.status <> 65535)THEN
					SDOWrite.enable	:= 0;
					SDO_wr			:= 0;
				END_IF
			END_IF

		4:
			DIO_Conf		:= 0;

			SDOWrite.pData		:= ADR(DIO_Conf);
			SDOWrite.datalen 	:= 2; //Data length, 2 bytes for 16-bit parameter
			SDOWrite.index 		:= 16#2008; //Index = 0x2000 + Menu Number
			SDOWrite.subindex	:= 23;
			SDOWrite.enable		:= 1;
			dlycnt1				:= dlycnt1 + 1;
			IF(dlycnt1 > 1)THEN
				IF (SDOWrite.status = 0) THEN
					SDOWrite.enable	:= 0;
					wr_step			:= 5;
					dlycnt1			:= 0;
					//				ELSIF((SDOWrite.status <> 65535)AND(SDOWrite.status <> 65534))THEN
				ELSIF(SDOWrite.status <> 65535)THEN
					SDOWrite.enable	:= 0;
					SDO_wr			:= 0;
				END_IF
			END_IF

		5:
			DIO_Conf		:= 0;

			SDOWrite.pData		:= ADR(DIO_Conf);
			SDOWrite.datalen 	:= 2; //Data length, 2 bytes for 16-bit parameter
			SDOWrite.index 		:= 16#2008; //Index = 0x2000 + Menu Number
			SDOWrite.subindex	:= 24;
			SDOWrite.enable		:= 1;
			dlycnt1				:= dlycnt1 + 1;
			IF(dlycnt1 > 1)THEN
				IF (SDOWrite.status = 0) THEN
					SDOWrite.enable	:= 0;
					wr_step			:= 6;
					dlycnt1			:= 0;
				ELSIF(SDOWrite.status <> 65535)THEN
					SDOWrite.enable	:= 0;
					SDO_wr			:= 0;
				END_IF
			END_IF

		6:
			//Enable the Control Word once configured

			Control_Enable		:= 1;
			SDOWrite.pData		:= ADR(Control_Enable);
			SDOWrite.datalen 	:= 1; //Data length, 2 bytes for 16-bit parameter
			SDOWrite.index 		:= 16#2006;
			SDOWrite.subindex	:= 43;
			SDOWrite.enable		:= 1;
			dlycnt1				:= dlycnt1 + 1;
			IF(dlycnt1 > 1)THEN
				IF (SDOWrite.status = 0) THEN
					SDOWrite.enable	:= 0;
					wr_step			:= 0;
					dlycnt1			:= 0;
					SDO_wr			:= 0;
					init			:= 0;
					SDO_rd			:= 1;
					execonce_wr		:= 1;
				ELSIF(SDOWrite.status <> 65535)THEN
					SDOWrite.enable	:= 0;
					SDO_wr			:= 0;
				END_IF
			END_IF

	END_CASE

	(* Once the Control word is configured on Power ON, read the status of the drive *)

	(* Reconfirm that the drives are in Run Mode & Control is enabled *)

	CASE rd_step OF
		0:
			IF((SDO_rd = 1)AND(DO1[0] = 1))THEN
				rd_step		:= 1;
				dlycnt		:= 0;
				Drv_Status	:= 0;
			END_IF
		1:
			// Reconfirm if Status Word still shows drive as Healty

			SDORead1.pData := ADR(Status_WORD); //Data to be read into here
			SDORead1.datalen := 2; //Data length, 2 bytes for 16-bit parameter
			SDORead1.index 		:= 16#200A;
			SDORead1.subindex	:= 40;
			SDORead1.enable		:= 1;
			dlycnt				:= dlycnt + 1;
			IF(dlycnt > 1)THEN
				IF (SDORead1.status = 0) THEN
					SDORead1.enable				:= 0;
					rd_step						:= 2;
					dlycnt						:= 0;
					Drv_Status					:= Status_WORD;
					Wind.Drive.Drive_Enable		:= Status_WORD.1;

				ELSIF(SDORead1.status <> 65535)THEN
					SDORead1.enable	:= 0;
				END_IF
			END_IF

		2:
			// Reconfirm if Control Word Enable is still 1

			SDORead1.pData 		:= ADR(Status_WORD); //Data to be read into here
			SDORead1.datalen 	:= 1; //Data length, 2 bytes for 16-bit parameter
			SDORead1.index 		:= 16#2006;
			SDORead1.subindex	:= 43;
			SDORead1.enable		:= 1;
			dlycnt				:= dlycnt + 1;
			IF(dlycnt > 1)THEN
				IF (SDORead1.status = 0) THEN
					SDORead1.enable	:= 0;
					rd_step			:= 0;
					dlycnt			:= 0;
					SDO_rd			:= 0;
					execonce_rd		:= 1;
					Control_Enb		:=	INT_TO_USINT(Status_WORD);
				ELSIF(SDORead1.status <> 65535)THEN
					SDORead1.enable	:= 0;
				END_IF
			END_IF
	END_CASE

	(* Disbale SDO read/write once the configuration is done *)
	IF((SDO_rd = 0)AND(execonce_rd = 1))THEN
		SDORead1.enable	:= 0;
		rd_step			:= 0;
		dlycnt			:= 0;
		execonce_rd		:= 0;
	END_IF

	IF((SDO_wr = 0)AND(init = 0)AND(execonce_wr = 1))THEN
		SDOWrite.enable	:= 0;
		wr_step			:= 0;
		dlycnt1			:= 0;
		execonce_wr		:= 0;
	END_IF

	(* AFter Power On, if the SDO Write is triggered then it is to Enable/Disable the drive.
	This enable/Disable is done by forcing the Control_Enable Bit *)

	IF((SDO_wr = 1)AND(init = 0))THEN
		//Control_Enable	:= 0;
		SDOWrite.pData		:= ADR(Control_Enable);
		SDOWrite.datalen 	:= 1; //Data length, 2 bytes for 16-bit parameter
		SDOWrite.index 		:= 16#2006;
		SDOWrite.subindex	:= 43;
		SDOWrite.enable		:= 1;
		dlycnt1				:= dlycnt1 + 1;
		IF(dlycnt1 > 1)THEN
			IF (SDOWrite.status = 0) THEN
				SDOWrite.enable	:= 0;
				wr_step			:= 0;
				dlycnt1			:= 0;
				SDO_wr			:= 0;
				SDO_rd			:= 1;
			ELSIF(SDOWrite.status <> 65535)THEN
				SDOWrite.enable	:= 0;
				SDO_wr			:= 0;
			END_IF
		END_IF
	END_IF

	IF((DigInp.Production_mode = 0)AND(DigInp.Jog_mode = 0)AND(statechg = 1))THEN
		Control_Enable	:= 0;
		SDO_wr			:= 1;
		statechg		:= 0;
	ELSIF((DigInp.Production_mode = 1)OR(DigInp.Jog_mode = 1)AND(statechg = 0))THEN
		statechg		:= 1;
		Control_Enable	:= 1;
		SDO_wr			:= 1;
	END_IF

	SDORead1();
	SDOWrite();

END_PROGRAM
```

#### Init.st
```iecst
PROGRAM _INIT
	(* Insert code here *)
	(* Insert code here *)
	(* Get NMT Status *)
	SDORead1.enable	:= 0;
	SDORead1.pDevice := ADR(PLC_INTF); //POWERLINK interface on MN (PLC) ‘IF1’
	SDORead1.node := 4; //Node address is set to 3

	SDOWrite.enable		:= 0;
	SDOWrite.node		:= 4;
	SDOWrite.pDevice	:= ADR(PLC_INTF);
	SDOWrite.pData		:= ADR(Control_WORD);

	DataReceived	:= 25;
	cnt_enable		:= 0;
	SDO_rdinit		:= 1;
	SDO_rd			:= 0;
	execonce_rd		:= 1;
	init			:= 1;
	SDO_wr			:= 0;
	execonce_wr		:= 0;
	dlycnt			:= 0;
	dlycnt1			:= 0;

END_PROGRAM
```

### Program Logical/EPLCom/Mot_Tun (IEC)

#### Variables.var
```iecst
VAR
	Control_Enable : SINT;
	dlycnt1 : USINT;
	Old_AxisMotor : INT;
	Old_AxisMotorTune : USINT;
	plc_node : USINT := 3;
	SDOMotor1_rd : EplSDORead;
	SDOMotor1_wr : EplSDOWrite;
	SDOMotor2_rd : EplSDORead;
	SDOMotor2_wr : EplSDOWrite;
	SDOTune_rd : EplSDORead;
	SDOTune_wr : EplSDOWrite;
	SDOWrite : EplSDOWrite;
	wr_step : USINT;
	Status_WORD : INT;
	dlycnt : USINT;
	Tune_Start : SINT;
	chkdly : USINT;
	firstchck : BOOL := FALSE;
	CopytoDrv : BOOL;
	motordata_step : USINT := 0;
END_VAR
```

#### Cyclic.st
```iecst
PROGRAM _CYCLIC
	(* Insert code here *)
	IF ( Save = 1 ) THEN
		CASE Axis_Motor OF
			0: 		// None

			1:		// Unwinder
				UnWind.MotorRating.RatedFreq 	:= TempFreq;
				UnWind.MotorRating.RatedCurrent := TempCurrent;
				UnWind.MotorRating.RatedVoltage := TempVoltage;
				UnWind.MotorRating.RatedSpeed	:= TempSpeed;
				UnWind.MotorRating.RatedPF 		:= TempPF;
				CopytoDrv						:= 1;
				plc_node						:= 3;

			2:		// Winder
				Wind.MotorRating.RatedFreq 		:= TempFreq;
				Wind.MotorRating.RatedCurrent 	:= TempCurrent;
				Wind.MotorRating.RatedVoltage 	:= TempVoltage;
				Wind.MotorRating.RatedSpeed		:= TempSpeed;
				Wind.MotorRating.RatedPF 		:= TempPF;
				CopytoDrv						:= 1;
				plc_node						:= 4;

			3:		// Infeed

			4:		// Outfeed

			5:		// Main

		END_CASE
		Save		:= 0;
		Axis_Motor	:= 0;
		Old_AxisMotor	:= Axis_Motor;
	ELSE
		IF(Axis_Motor <> Old_AxisMotor)THEN
			CASE Axis_Motor OF
				0: 		// None
					TempFreq	:= 0;
					TempCurrent	:= 0;
					TempVoltage	:= 0;
					TempSpeed	:= 0;
					TempPF		:= 0;

				1:		// Unwinder
					TempFreq	:= UnWind.MotorRating.RatedFreq;
					TempCurrent	:= UnWind.MotorRating.RatedCurrent;
					TempVoltage	:= UnWind.MotorRating.RatedVoltage;
					TempSpeed	:= UnWind.MotorRating.RatedSpeed;
					TempPF		:= UnWind.MotorRating.RatedPF;

				2:		// Winder
					TempFreq	:= Wind.MotorRating.RatedFreq;
					TempCurrent	:= Wind.MotorRating.RatedCurrent;
					TempVoltage	:= Wind.MotorRating.RatedVoltage;
					TempSpeed	:= Wind.MotorRating.RatedSpeed;
					TempPF		:= Wind.MotorRating.RatedPF;

				3:		// Infeed
					TempFreq	:= 0;
					TempCurrent	:= 0;
					TempVoltage	:= 0;
					TempSpeed	:= 0;
					TempPF		:= 0;

				4:		// Outfeed
					TempFreq	:= 0;
					TempCurrent	:= 0;
					TempVoltage	:= 0;
					TempSpeed	:= 0;
					TempPF		:= 0;

				5:		// Main
					TempFreq	:= 0;
					TempCurrent	:= 0;
					TempVoltage	:= 0;
					TempSpeed	:= 0;
					TempPF		:= 0;

			END_CASE
			Old_AxisMotor	:= Axis_Motor;
		END_IF
	END_IF

	CASE motordata_step OF
		0:
			IF(CopytoDrv = 1)THEN
				motordata_step	:= 1;
				dlycnt1			:= 0;
			END_IF

		1:
			SDOWrite.node		:= plc_node;
			SDOWrite.pData		:= ADR(TempFreq);
			SDOWrite.datalen 	:= 4; //Data length, 2 bytes for 16-bit parameter
			SDOWrite.index 		:= 16#2005;
			SDOWrite.subindex	:= 6;
			SDOWrite.enable		:= 1;
			dlycnt1				:= dlycnt1 + 1;
			IF(dlycnt1 > 1)THEN
				IF (SDOWrite.status = 0) THEN
					SDOWrite.enable	:= 0;
					motordata_step	:= 2;
					dlycnt1			:= 0;
				ELSIF(SDOWrite.status <> 65535)THEN
					SDOWrite.enable	:= 0;
					motordata_step	:= 0;
					CopytoDrv		:= 0;
				END_IF
			END_IF

		2:
			// Write Motor Current
			SDOWrite.node		:= plc_node;
			SDOWrite.pData		:= ADR(TempCurrent);
			SDOWrite.datalen 	:= 4; //Data length, 2 bytes for 16-bit parameter
			SDOWrite.index 		:= 16#2005;
			SDOWrite.subindex	:= 7;
			SDOWrite.enable		:= 1;
			dlycnt1				:= dlycnt1 + 1;
			IF(dlycnt1 > 1)THEN
				IF (SDOWrite.status = 0) THEN
					SDOWrite.enable	:= 0;
					motordata_step	:= 3;
					dlycnt1			:= 0;
				ELSIF(SDOWrite.status <> 65535)THEN
					SDOWrite.enable	:= 0;
					motordata_step	:= 0;
					CopytoDrv		:= 0;
				END_IF
			END_IF

		3:
			SDOWrite.node		:= plc_node;
			SDOWrite.pData		:= ADR(TempVoltage);
			SDOWrite.datalen 	:= 2; //Data length, 2 bytes for 16-bit parameter
			SDOWrite.index 		:= 16#2005; //Index = 0x2000 + Menu Number
			SDOWrite.subindex	:= 9;
			SDOWrite.enable		:= 1;
			dlycnt1				:= dlycnt1 + 1;
			IF(dlycnt1 > 1)THEN
				IF (SDOWrite.status = 0) THEN
					SDOWrite.enable	:= 0;
					motordata_step	:= 4;
					dlycnt1			:= 0;
				ELSIF(SDOWrite.status <> 65535)THEN
					SDOWrite.enable	:= 0;
					motordata_step	:= 0;
					CopytoDrv		:= 0;
				END_IF
			END_IF

		4:
			SDOWrite.node		:= plc_node;
			SDOWrite.pData		:= ADR(TempSpeed);
			SDOWrite.datalen 	:= 4; //Data length, 2 bytes for 16-bit parameter
			SDOWrite.index 		:= 16#2005; //Index = 0x2000 + Menu Number
			SDOWrite.subindex	:= 8;
			SDOWrite.enable		:= 1;
			dlycnt1				:= dlycnt1 + 1;
			IF(dlycnt1 > 1)THEN
				IF (SDOWrite.status = 0) THEN
					SDOWrite.enable	:= 0;
					motordata_step	:= 5;
					dlycnt1			:= 0;
				ELSIF(SDOWrite.status <> 65535)THEN
					SDOWrite.enable	:= 0;
					motordata_step	:= 0;
					CopytoDrv		:= 0;
				END_IF
			END_IF
		5:
			SDOWrite.node		:= plc_node;
			SDOWrite.pData		:= ADR(TempPF);
			SDOWrite.datalen 	:= 2; //Data length, 2 bytes for 16-bit parameter
			SDOWrite.index 		:= 16#2005; //Index = 0x2000 + Menu Number
			SDOWrite.subindex	:= 10;
			SDOWrite.enable		:= 1;
			dlycnt1				:= dlycnt1 + 1;
			IF(dlycnt1 > 1)THEN
				IF (SDOWrite.status = 0) THEN
					SDOWrite.enable	:= 0;
					motordata_step	:= 0;
					dlycnt1			:= 0;
					CopytoDrv		:= 0;
				ELSIF(SDOWrite.status <> 65535)THEN
					SDOWrite.enable	:= 0;
					motordata_step	:= 0;
					CopytoDrv		:= 0;
				END_IF
			END_IF
	END_CASE

	IF(Tune_Enable = 1)THEN
		Old_AxisMotorTune	:= Axis_MotorTune;
	END_IF

	(* Initial Power Up Configuring the Control Word to Read Freq. Command from Preset-1 & disable other preset values
	& enable the Control *)

	CASE wr_step OF
		0:
			IF(Tune_Enable = 1)THEN
				IF(Axis_MotorTune = 1)THEN
					plc_node	:= 3;
				ELSIF(Axis_MotorTune = 2)THEN
					plc_node	:= 4;
				END_IF
				wr_step		:= 1; //Tune UnWinder motor
				dlycnt	:= 0;
			END_IF

		1:
			//Disable the Control Enable
			Control_Enable		:= 0;

			SDOTune_wr.node		:= plc_node;
			SDOTune_wr.pData	:= ADR(Control_Enable);
			SDOTune_wr.datalen 	:= 1; //Data length, 2 bytes for 16-bit parameter
			SDOTune_wr.index 	:= 16#2006;
			SDOTune_wr.subindex	:= 43;
			SDOTune_wr.enable	:= 1;
			dlycnt				:= dlycnt + 1;
			IF(dlycnt > 1)THEN
				IF (SDOTune_wr.status = 0) THEN
					SDOTune_wr.enable	:= 0;
					wr_step				:= 2;
					dlycnt				:= 0;
				ELSIF(SDOTune_wr.status <> 65535)THEN
					SDOTune_wr.enable	:= 0;
				END_IF
			END_IF
		2:
			//Confirm that the Drive is not Active

			SDOTune_rd.node		:= plc_node;
			SDOTune_rd.pData 	:= ADR(Status_WORD); //Data to be read into here
			SDOTune_rd.datalen	:= 2; //Data length, 2 bytes for 16-bit parameter
			SDOTune_rd.index 	:= 16#200A;
			SDOTune_rd.subindex	:= 40;
			SDOTune_rd.enable	:= 1;
			dlycnt				:= dlycnt + 1;
			IF(dlycnt > 1)THEN
				IF (SDOTune_rd.status = 0) THEN
					SDOTune_rd.enable	:= 0;
					dlycnt				:= 0;
					IF(Status_WORD.1 = 0)THEN
						wr_step			:= 3;
					END_IF
				ELSIF(SDOTune_rd.status <> 65535)THEN
					SDOTune_rd.enable	:= 0;
				END_IF
			END_IF

		3:
			// Set the Auto Tune Bit
			Tune_Start			:= 2;

			SDOTune_wr.pData	:= ADR(Tune_Start);
			SDOTune_wr.datalen 	:= 1; //Data length, 2 bytes for 16-bit parameter
			SDOTune_wr.index 	:= 16#2005;
			SDOTune_wr.subindex	:= 12;
			SDOTune_wr.enable	:= 1;
			dlycnt				:= dlycnt + 1;
			IF(dlycnt > 3)THEN
				IF (SDOTune_wr.status = 0) THEN
					SDOTune_wr.enable	:= 0;
					wr_step			:= 4;
					dlycnt			:= 0;
					firstchck		:= 1;
				ELSIF(SDOTune_wr.status <> 65535)THEN
					SDOTune_wr.enable	:= 0;
				END_IF
			END_IF
		4:
			//Disable the Control Enable
			Control_Enable		:= 1;

			SDOTune_wr.node		:= plc_node;
			SDOTune_wr.pData	:= ADR(Control_Enable);
			SDOTune_wr.datalen 	:= 1; //Data length, 2 bytes for 16-bit parameter
			SDOTune_wr.index 	:= 16#2006;
			SDOTune_wr.subindex	:= 43;
			SDOTune_wr.enable	:= 1;
			dlycnt				:= dlycnt + 1;
			IF(dlycnt > 1)THEN
				IF (SDOTune_wr.status = 0) THEN
					SDOTune_wr.enable	:= 0;
					wr_step				:= 5;
					dlycnt				:= 0;
				ELSIF(SDOTune_wr.status <> 65535)THEN
					SDOTune_wr.enable	:= 0;
				END_IF
			END_IF

		5:
			// Check if Auto Tune is complete
			SDOTune_rd.node		:= plc_node;
			SDOTune_rd.pData 	:= ADR(Status_WORD);
			SDOTune_rd.datalen	:= 1;
			SDOTune_rd.index 	:= 16#2005;
			SDOTune_rd.subindex	:= 12;

			IF(firstchck = 1)THEN
				SDOTune_rd.enable	:= 1;
			ELSIF(chkdly > 50)THEN
				SDOTune_rd.enable	:= 1;
				chkdly				:= 0;
			END_IF

			dlycnt			:= dlycnt + 1;

			IF(dlycnt > 1)THEN
				IF (SDOTune_rd.status = 0) THEN
					SDOTune_rd.enable	:= 0;
					IF(Status_WORD = 0)THEN
						wr_step		:= 0;
						Tune_Enable	:= 0;
						dlycnt		:= 0;
						chkdly		:= 0;
					END_IF
				ELSIF(SDOTune_rd.status <> 65535)THEN
					SDOTune_rd.enable	:= 0;
				END_IF
			END_IF

			IF(Status_WORD = 2)THEN
				chkdly	:= chkdly + 1;
			END_IF

	END_CASE

	SDOTune_wr();
	SDOTune_rd();
	SDOWrite();

END_PROGRAM
```

### Program Logical/EPLCom/TunePID (IEC)

#### Variables.var
```iecst
VAR
	SDORead_PID : EplSDORead;
	SDO_PIDWR : EplSDOWrite;
	dlycnt_wrpid : USINT;
	wrpid_step : USINT;
	SDO_pidwr : BOOL;
	dlycnt_pid : USINT;
	rdpid_step : USINT;
	SDO_pid : BOOL;
	PID_RefSrc : INT;
	RefSrc_WORD : INT;
	Derv_Gain : INT;
	PID_WORD : INT;
	Ingr_Gain : INT;
	Porp_Gain : INT;
	SDO_wr : BOOL;
	RefSrc_Set : INT;
	DerGain_Set : INT;
	IntGain_Set : INT;
	PropGain_Set : INT;
	CopytoDrv : BOOL;
	plc_node : USINT;
	Old_AxisMotor : INT;
	SDOWrite_PID : EplSDOWrite;
	Axis_PID : USINT;
	TempUpperLim : INT;
	TempLowerLim : INT;
	TempPIDEnable : USINT;
	Old_AxisPID : USINT;
END_VAR
```

#### Cyclic.st
```iecst
PROGRAM _CYCLIC
    (* Write the PID values to the Drive as well as write Reference Source and Destination Addresses *)
	IF ( SavePID = 1 ) THEN
		CASE Axis_PID OF
			0: 		// None

			1:		// Unwinder
				UnWind.Tension.PID.Prop_Gain 		:= TempPropGain;
				UnWind.Tension.PID.Intg_Gain 		:= TempIntgGain;
				UnWind.Tension.PID.Derv_Gain 		:= TempDervGain;
				UnWind.Tension.PID.Reference_Add	:= TempPIDRef;
				UnWind.Tension.PID.Feedback_Add		:= TempPIDFeedback;
				UnWind.Tension.PID.Enable			:= TempPIDEnable;
				UnWind.Tension.PID.UpperLimit		:= TempUpperLim;
				UnWind.Tension.PID.LowerLimit		:= TempLowerLim;

				CopytoDrv	:= 1;
				plc_node	:= 3;
				SDO_pidwr	:= 1; // Trigger the PID Write State Machine

			2:		// Winder
				Wind.Tension.PID.Prop_Gain 		:= TempPropGain;
				Wind.Tension.PID.Intg_Gain 		:= TempIntgGain;
				Wind.Tension.PID.Derv_Gain 		:= TempDervGain;
				Wind.Tension.PID.Reference_Add	:= TempPIDRef;
				Wind.Tension.PID.Feedback_Add	:= TempPIDFeedback;
				Wind.Tension.PID.Enable			:= TempPIDEnable;
				Wind.Tension.PID.UpperLimit		:= TempUpperLim;
				Wind.Tension.PID.LowerLimit		:= TempLowerLim;

				CopytoDrv	:= 1;
				plc_node	:= 4;
				SDO_pidwr	:= 1; // Trigger the PID Write State Machine

			3:		// Infeed

			4:		// Outfeed

			5:		// Main

		END_CASE
		SavePID			:= 0;
		Axis_PID		:= 0;
		Old_AxisPID		:= Axis_PID;

	ELSE
		IF(Axis_PID <> Old_AxisPID)THEN
			CASE Axis_PID OF
				0: 		// None
					TempPropGain	:= 0;
					TempIntgGain	:= 0;
					TempDervGain	:= 0;
					TempPIDRef		:= 0;
					TempPIDFeedback := 0;
					TempPIDEnable	:= 0;
					TempUpperLim	:= 0;
					TempLowerLim	:= 0;

				1:		// Unwinder
					TempPropGain	:= UnWind.Tension.PID.Prop_Gain;
					TempIntgGain	:= UnWind.Tension.PID.Intg_Gain;
					TempDervGain	:= UnWind.Tension.PID.Derv_Gain;
					TempPIDRef		:= UnWind.Tension.PID.Reference_Add;
					TempPIDFeedback	:= UnWind.Tension.PID.Feedback_Add;
					TempPIDEnable	:= UnWind.Tension.PID.Enable;
					TempUpperLim	:= UnWind.Tension.PID.UpperLimit;
					TempLowerLim	:= UnWind.Tension.PID.LowerLimit;

				2:		// Winder
					TempPropGain	:= Wind.Tension.PID.Prop_Gain;
					TempIntgGain	:= Wind.Tension.PID.Intg_Gain;
					TempDervGain	:= Wind.Tension.PID.Derv_Gain;
					TempPIDRef		:= Wind.Tension.PID.Reference_Add;
					TempPIDFeedback	:= Wind.Tension.PID.Feedback_Add;
					TempPIDEnable	:= Wind.Tension.PID.Enable;
					TempUpperLim	:= Wind.Tension.PID.UpperLimit;
					TempLowerLim	:= Wind.Tension.PID.LowerLimit;

				3:		// Infeed
					TempPropGain	:= 0;
					TempIntgGain	:= 0;
					TempDervGain	:= 0;
					TempPIDRef		:= 0;
					TempPIDFeedback	:= 0;
					TempPIDEnable	:= 0;
					TempUpperLim	:= 0;
					TempLowerLim	:= 0;

				4:		// Outfeed
					TempPropGain	:= 0;
					TempIntgGain	:= 0;
					TempDervGain	:= 0;
					TempPIDRef		:= 0;
					TempPIDFeedback	:= 0;
					TempPIDEnable	:= 0;
					TempUpperLim	:= 0;
					TempLowerLim	:= 0;

				5:		// Main
					TempPropGain	:= 0;
					TempIntgGain	:= 0;
					TempDervGain	:= 0;
					TempPIDRef		:= 0;
					TempPIDFeedback := 0;
					TempPIDEnable	:= 0;
					TempUpperLim	:= 0;
					TempLowerLim	:= 0;

			END_CASE
			Old_AxisPID		:= Axis_PID;
		END_IF
	END_IF

	CASE wrpid_step OF
		0: // Idle - Wait for trigger
			IF(SDO_pidwr = 1)THEN
				wrpid_step		:= 1;
				dlycnt_wrpid	:= 0;
			END_IF

		1: // Write Proportional Gain
			SDO_PIDWR.node		:= plc_node; // <- CRITICAL: Set the node address
			SDO_PIDWR.pData		:= ADR(TempPropGain); // Write the Temp value from UI
			SDO_PIDWR.datalen 	:= 2;
			SDO_PIDWR.index 	:= 16#200E;
			SDO_PIDWR.subindex	:= 10;
			SDO_PIDWR.enable	:= 1;
			dlycnt_wrpid		:= dlycnt_wrpid + 1;

			IF(dlycnt_wrpid > 1)THEN
				IF (SDO_PIDWR.status = 0) THEN
					SDO_PIDWR.enable	:= 0;
					wrpid_step			:= 2;
					dlycnt_wrpid		:= 0;
				ELSIF(SDO_PIDWR.status <> 65535)THEN // If any other error occurs
					SDO_PIDWR.enable	:= 0;
					wrpid_step			:= 0; // Reset state machine on error
					dlycnt_wrpid		:= 0;
					SDO_pidwr			:= 0;
				END_IF
			END_IF

		2: // Write Integral Gain
			SDO_PIDWR.node		:= plc_node;
			SDO_PIDWR.pData		:= ADR(TempIntgGain);
			SDO_PIDWR.datalen 	:= 2;
			SDO_PIDWR.index 	:= 16#200E;
			SDO_PIDWR.subindex	:= 11;
			SDO_PIDWR.enable	:= 1;
			dlycnt_wrpid		:= dlycnt_wrpid + 1;

			IF(dlycnt_wrpid > 1)THEN
				IF (SDO_PIDWR.status = 0) THEN
					SDO_PIDWR.enable	:= 0;
					wrpid_step			:= 3;
					dlycnt_wrpid		:= 0;
				ELSIF(SDO_PIDWR.status <> 65535)THEN
					SDO_PIDWR.enable	:= 0;
					wrpid_step			:= 0;
					dlycnt_wrpid		:= 0;
					SDO_pidwr			:= 0;
				END_IF
			END_IF

		3: // Write Derivative Gain
			SDO_PIDWR.node		:= plc_node;
			SDO_PIDWR.pData		:= ADR(TempDervGain);
			SDO_PIDWR.datalen 	:= 2;
			SDO_PIDWR.index 	:= 16#200E;
			SDO_PIDWR.subindex	:= 12;
			SDO_PIDWR.enable	:= 1;
			dlycnt_wrpid		:= dlycnt_wrpid + 1;

			IF(dlycnt_wrpid > 1)THEN
				IF (SDO_PIDWR.status = 0) THEN
					SDO_PIDWR.enable	:= 0;
					wrpid_step			:= 4;
					dlycnt_wrpid		:= 0;
				ELSIF(SDO_PIDWR.status <> 65535)THEN
					SDO_PIDWR.enable	:= 0;
					wrpid_step			:= 0;
					dlycnt_wrpid		:= 0;
					SDO_pidwr			:= 0;
				END_IF
			END_IF

		4: // Write Reference Source (Optional Configuration)
			SDO_PIDWR.node		:= plc_node;
			SDO_PIDWR.pData		:= ADR(TempPIDRef); // Assuming this is set elsewhere
			SDO_PIDWR.datalen 	:= 2;
			SDO_PIDWR.index 	:= 16#200E;
			SDO_PIDWR.subindex	:= 03;	// This is linked to 12.008
			SDO_PIDWR.enable	:= 1;
			dlycnt_wrpid		:= dlycnt_wrpid + 1;

			IF(dlycnt_wrpid > 1)THEN
				IF (SDO_PIDWR.status = 0) THEN
					SDO_PIDWR.enable	:= 0;
					wrpid_step			:= 5;
					dlycnt_wrpid		:= 0;
				ELSIF(SDO_PIDWR.status <> 65535)THEN
					SDO_PIDWR.enable	:= 0;
					wrpid_step			:= 0;
					dlycnt_wrpid		:= 0;
					SDO_pidwr			:= 0;
				END_IF
			END_IF

		5: // Write Feedback Source (Optional Configuration)
			SDO_PIDWR.node		:= plc_node;
			SDO_PIDWR.pData		:= ADR(TempPIDFeedback); // Assuming this is set elsewhere
			SDO_PIDWR.datalen 	:= 2;
			SDO_PIDWR.index 	:= 16#200E;
			SDO_PIDWR.subindex	:= 04;	// This is linked to 7.001
			SDO_PIDWR.enable	:= 1;
			dlycnt_wrpid		:= dlycnt_wrpid + 1;

			IF(dlycnt_wrpid > 1)THEN
				IF (SDO_PIDWR.status = 0) THEN
					SDO_PIDWR.enable	:= 0;
					wrpid_step			:= 6;
					dlycnt_wrpid		:= 0;
				ELSIF(SDO_PIDWR.status <> 65535)THEN
					SDO_PIDWR.enable	:= 0;
					wrpid_step			:= 0;
					dlycnt_wrpid		:= 0;
					SDO_pidwr			:= 0;
				END_IF
			END_IF
		6: // Write Output Upper Limit (Optional Configuration)
			SDO_PIDWR.node		:= plc_node;
			SDO_PIDWR.pData		:= ADR(TempUpperLim); // Assuming this is set elsewhere
			SDO_PIDWR.datalen 	:= 2;
			SDO_PIDWR.index 	:= 16#200E;
			SDO_PIDWR.subindex	:= 13;
			SDO_PIDWR.enable	:= 1;
			dlycnt_wrpid		:= dlycnt_wrpid + 1;

			IF(dlycnt_wrpid > 1)THEN
				IF (SDO_PIDWR.status = 0) THEN
					SDO_PIDWR.enable	:= 0;
					wrpid_step			:= 7;
					dlycnt_wrpid		:= 0;
				ELSIF(SDO_PIDWR.status <> 65535)THEN
					SDO_PIDWR.enable	:= 0;
					wrpid_step			:= 0;
					dlycnt_wrpid		:= 0;
					SDO_pidwr			:= 0;
				END_IF
			END_IF

		7: // Write Output Lower Limit (Optional Configuration)
			SDO_PIDWR.node		:= plc_node;
			SDO_PIDWR.pData		:= ADR(TempLowerLim); // Assuming this is set elsewhere
			SDO_PIDWR.datalen 	:= 2;
			SDO_PIDWR.index 	:= 16#200E;
			SDO_PIDWR.subindex	:= 14;
			SDO_PIDWR.enable	:= 1;
			dlycnt_wrpid		:= dlycnt_wrpid + 1;

			IF(dlycnt_wrpid > 1)THEN
				IF (SDO_PIDWR.status = 0) THEN
					SDO_PIDWR.enable	:= 0;
					wrpid_step			:= 8;
					dlycnt_wrpid		:= 0;
				ELSIF(SDO_PIDWR.status <> 65535)THEN
					SDO_PIDWR.enable	:= 0;
					wrpid_step			:= 0;
					dlycnt_wrpid		:= 0;
					SDO_pidwr			:= 0;
				END_IF
			END_IF

		8: // Write PID Enable/Disable
			SDO_PIDWR.node		:= plc_node;
			SDO_PIDWR.pData		:= ADR(TempPIDEnable); // Assuming this is set elsewhere
			SDO_PIDWR.datalen 	:= 1;
			SDO_PIDWR.index 	:= 16#200E;
			SDO_PIDWR.subindex	:= 08;
			SDO_PIDWR.enable	:= 1;
			dlycnt_wrpid		:= dlycnt_wrpid + 1;

			IF(dlycnt_wrpid > 1)THEN
				IF (SDO_PIDWR.status = 0) THEN
					SDO_PIDWR.enable	:= 0;
					wrpid_step			:= 0;
					dlycnt_wrpid		:= 0;
					SDO_pidwr			:= 0;
				ELSIF(SDO_PIDWR.status <> 65535)THEN
					SDO_PIDWR.enable	:= 0;
					wrpid_step			:= 0;
					dlycnt_wrpid		:= 0;
					SDO_pidwr			:= 0;
				END_IF
			END_IF

	END_CASE

(*
	CASE rdpid_step OF
		0: // Idle - Wait for trigger
			IF(SDO_pid = 1)THEN
				rdpid_step	:= 1;
				dlycnt_pid	:= 0;
			END_IF

		1: // Read Proportional Gain
			SDORead_PID.node		:= plc_node; // <- CRITICAL: Set the node address
			SDORead_PID.pData 		:= ADR(PID_WORD);
			SDORead_PID.datalen 	:= 2;
			SDORead_PID.index 		:= 16#200E;
			SDORead_PID.subindex	:= 10;
			SDORead_PID.enable		:= 1;
			dlycnt_pid				:= dlycnt_pid + 1;

			IF(dlycnt_pid > 2)THEN
				IF (SDORead_PID.status = 0) THEN
					SDORead_PID.enable	:= 0;
					rdpid_step			:= 2;
					dlycnt_pid			:= 0;
					UnWind.Tension.PID.Prop_Gain	:= PID_WORD; // Store read value
				ELSIF(SDORead_PID.status <> 65535)THEN
					SDORead_PID.enable	:= 0;
					rdpid_step			:= 0; // Reset on error
					dlycnt_pid			:= 0;
					SDO_pid				:= 0;
				END_IF
			END_IF

		2: // Read Integral Gain
			SDORead_PID.node		:= plc_node;
			SDORead_PID.pData 		:= ADR(PID_WORD);
			SDORead_PID.datalen 	:= 2;
			SDORead_PID.index 		:= 16#200E;
			SDORead_PID.subindex	:= 11;
			SDORead_PID.enable		:= 1;
			dlycnt_pid				:= dlycnt_pid + 1;

			IF(dlycnt_pid > 2)THEN
				IF (SDORead_PID.status = 0) THEN
					SDORead_PID.enable	:= 0;
					rdpid_step			:= 3;
					dlycnt_pid			:= 0;
					UnWind.Tension.PID.Intg_Gain	:= PID_WORD;
				ELSIF(SDORead_PID.status <> 65535)THEN
					SDORead_PID.enable	:= 0;
					rdpid_step			:= 0;
					dlycnt_pid			:= 0;
					SDO_pid				:= 0;
				END_IF
			END_IF

		3: // Read Derivative Gain
			SDORead_PID.node		:= plc_node;
			SDORead_PID.pData 		:= ADR(PID_WORD);
			SDORead_PID.datalen 	:= 2;
			SDORead_PID.index 		:= 16#200E;
			SDORead_PID.subindex	:= 12;
			SDORead_PID.enable		:= 1;
			dlycnt_pid				:= dlycnt_pid + 1;

			IF(dlycnt_pid > 2)THEN
				IF (SDORead_PID.status = 0) THEN
					SDORead_PID.enable	:= 0;
					rdpid_step			:= 4;
					dlycnt_pid			:= 0;
					UnWind.Tension.PID.Derv_Gain	:= PID_WORD;
				ELSIF(SDORead_PID.status <> 65535)THEN
					SDORead_PID.enable	:= 0;
					rdpid_step			:= 0;
					dlycnt_pid			:= 0;
					SDO_pid				:= 0;
				END_IF
			END_IF

		4: // Read Reference Source
			SDORead_PID.node		:= plc_node;
			SDORead_PID.pData 		:= ADR(RefSrc_WORD);
			SDORead_PID.datalen 	:= 2;
			SDORead_PID.index 		:= 16#200E;
			SDORead_PID.subindex	:= 03;
			SDORead_PID.enable		:= 1;
			dlycnt_pid				:= dlycnt_pid + 1;

			IF(dlycnt_pid > 2)THEN
				IF (SDORead_PID.status = 0) THEN
					SDORead_PID.enable	:= 0;
					rdpid_step			:= 0; // Sequence complete
					dlycnt_pid			:= 0;
					SDO_pid				:= 0; // Clear the trigger
					PID_RefSrc			:= INT_TO_UINT(RefSrc_WORD);
				ELSIF(SDORead_PID.status <> 65535)THEN
					SDORead_PID.enable	:= 0;
					rdpid_step			:= 0;
					dlycnt_pid			:= 0;
					SDO_pid				:= 0;
				END_IF
			END_IF
	END_CASE
  *)

	(* Safety Nets: Ensure state machines reset cleanly if their trigger is cleared externally *)
(*	IF(SDO_pid = 0)THEN
		SDORead_PID.enable	:= 0;
		rdpid_step			:= 0;
		dlycnt_pid			:= 0;
	END_IF
*)
	IF(SDO_pidwr = 0)THEN
		SDO_PIDWR.enable	:= 0;
		wrpid_step			:= 0;
		dlycnt_wrpid		:= 0;
	END_IF

	(* Execute the SDO function blocks *)
	SDO_PIDWR();
//	SDORead_PID();

END_PROGRAM
```

#### Init.st
```iecst
PROGRAM _INIT
	(* Insert code here *)
	SDORead_PID.enable	:= 0;
	SDORead_PID.pDevice := ADR(PLC_INTF); //POWERLINK interface on MN (PLC) ‘IF1’
	SDORead_PID.node := 3; //Node address is set to 3

	SDO_PIDWR.enable	:= 0;
	SDO_PIDWR.node		:= 3;
	SDO_PIDWR.pDevice	:= ADR(PLC_INTF);

	Axis_PID	:= 0;
	CopytoDrv	:= 0;
	plc_node	:= 3;
	SDO_pidwr	:= 0;
	SavePID		:= 0;
	Old_AxisPID	:= 0;
	dlycnt_wrpid := 0;

END_PROGRAM
```

### Program Logical/5Drive/HS_Inp (IEC)

#### Variables.var
```iecst
VAR
	ActInfeedKN : LCScINT;
	ActOutfeedKN : LCScINT;
	ActUnWindKN : LCScINT;
	ActUnWindRPM : LCLiScINT;
	i : USINT;
	Axis_RpmInpFilt : ARRAY[0..4] OF LCPT1;
	HSCounter : LCCounter;
	initialize : BOOL;
	MainRoleDia : INT;
	InfeedRoleDia : INT;
	OutfeedRoleDia : INT;
	Axis_KNInpFilt : ARRAY[0..4] OF LCPT1;
END_VAR
```

#### HS_Inp_Cyclic.st
```iecst
PROGRAM _CYCLIC

	(* Time base counter *)
	HSCounter();

	(*Used 4th Channel of AI2 for Winder RPM. Copy the same to the 5th element of array AI3 *)
	IF(initialize = 1)THEN
		(* Initialize filter of all axes to 0 *)
		FOR i := 0 TO (MAX_AXES - 1) DO
			Axis_RpmInpFilt[i].x := 0;
			Axis_RpmInpFilt[i]();
			AxisRPM[i].InpBits := Axis_RpmInpFilt[i].y;
		END_FOR

		(* Initialize filtRPM of all axes to 0 *)
		FOR i := 0 TO (MAX_AXES-1) DO
			Axis_RPM[i].x:= 0;
			Axis_RPM[i]();
		END_FOR

		FOR i := 0 TO (MAX_AXES - 1) DO
			Axis_KNInpFilt[i].x	:= 0;
			Axis_KNInpFilt[i]();
			AxisKN[i].InpBits := Axis_KNInpFilt[i].y;
		END_FOR

		(* Initialize filtRPM of all axes to 0 *)
		FOR i := 0 TO (MAX_AXES-1) DO
			Axis_KN[i].x := 0;
			Axis_KN[i]();
		END_FOR

		initialize := 0;

	ELSE

		(* CALCULATE RPM OF EACH AXIS *)

		(* Adding filter to analog inputs for RPM *)
		FOR i := 0 TO (MAX_AXES - 1) DO
			Axis_RpmInpFilt[i].x := AI3[i];
			Axis_RpmInpFilt[i]();

			AxisRPM[i].InpBits := Axis_RpmInpFilt[i].y;
		END_FOR

		FOR i := 0 TO (MAX_AXES-1) DO
			Axis_RPM[i].x := AxisRPM[i].InpBits;
			Axis_RPM[i]();
		END_FOR

		Actual.UnWindRPM	:= Axis_RPM[UNWINDER].y;
		Actual.InfeedRPM	:= Axis_RPM[INFEED].y;
		Actual.OutfeedRPM	:= Axis_RPM[OUTFEED].y;
		Actual.WindRPM		:= Axis_RPM[WINDER].y;

		(* CALCULATE ACTUAL RPM AND DIAMETER OF Winder/Unwinder *)
		Actual.RPM 	:= (Encoder_counts/PulsesPerRev) * 60

		(* CALCULATE MPM OF EACH AXIS *)
		Actual.MainMPM		:= (Actual.MainRPM * 314 * Set.MainRoleDia)/100; (* Main Roller MPM UNIT 0.001 *)

		Actual.UnWindDia	:= (Actual.MainMPM * 100)/(Actual.UnWindRPM * 314); (* UnWinder MPM UNIT 0.001 *)

		Actual.InfeedMPM	:= (Actual.InfeedRPM * 314 * Set.InfeedRolerDia)/100;(* InFeed MPM UNIT 0.001 *)

		Actual.OutfeedMPM	:= (Actual.OutfeedRPM * 314 * Set.OutfeedRolerDia)/100; (* OutFeed MPM UNIT 0.001 *)

		Actual.WindDia		:= (Actual.MainMPM * 100)/(Actual.WindRPM * 314);  (* Winder MPM UNIT 0.001 *)

		(* SCALE MPM OF EACH AXIS by FACTOR OF 1024 *)
		Actual.MainMPM		:=  (Actual.MainPulses * 314 * Set.MainRoleDia)/102400; (* Main Roller MPM UNIT 0.001 *)

		Actual.UnWindDia	:= (Actual.MainMPM * PulsesPerRev * 100)/(Actual.UnWindPulses * 314); (* UnWinder MPM UNIT 0.001 *)

		Actual.InfeedMPM	:= (Actual.InfeedPulses * 314 * Set.InfeedRolerDia)/PulsesPerRev * 100;(* InFeed MPM UNIT 0.001 *)

		Actual.OutfeedMPM	:= (Actual.OutfeedPulses * 314 * Set.OutfeedRolerDia)/PulsesPerRev * 100; (* OutFeed MPM UNIT 0.001 *)

		Actual.WindDia		:= (Actual.MainMPM * PulsesPerRev * 100)/(Actual.WindPulses * 314);  (* Winder MPM UNIT 0.001 *)

		Actual.WindDia := ((Actual.MPM * 100 )/(314 * Actual.RPM)) - Wind.Dia.MinDia;

		Actual.UnWindDia := ((Actual.MPM * 100 )/(314 * Actual.RPM)) + UnWind.Dia.MinDia;

		(* NUMBER OF REVOLUTIONS FROM SCALED MPM *)
		Actual.MainRevs 	:= Actual.MainPulses/PulsesPerRev;

		Actual.UnWindRevs 	:= Actual.UnWindPulses/PulsesPerRev;

		Actual.InfeedRevs 	:= Actual.InfeedPulses/PulsesPerRev;

		Actual.OutfeedRevs 	:= Actual.OutfeedPulses/PulsesPerRev;

		Actual.WindRevs 	:= Actual.WindPulses/PulsesPerRev;

		(* CALCULATE Tension(KN) OF EACH AXIS *)

		(* Adding filter to analog inputs for LoadCell *)

		FOR i := 0 TO (MAX_AXES - 1) DO
			Axis_KNInpFilt[i].x	:= AI1[i];
			Axis_KNInpFilt[i]();

			AxisKN[i].InpBits := Axis_KNInpFilt[i].y;
		END_FOR

		FOR i := 0 TO (MAX_AXES-1) DO
			Axis_KN[i].x := AxisKN[i].InpBits;
			Axis_KN[i]();
		END_FOR

		Actual.UnWindTension	:= Axis_KN[UNWINDER].y;
		Actual.InfeedTension	:= Axis_KN[INFEED].y;
		Actual.OutfeedTension	:= Axis_KN[OUTFEED].y;
		Actual.WindTension		:= Axis_KN[WINDER].y;

		Timer(IN := Enable, PT := T#2s);  // Start timer when Enable is TRUE

		// Rising edge detection for timer.Q
		IF (Timer.Q AND NOT Timer.IN) THEN
			SampledMPM := ActualMPM;
			SampledRPM := ActualRPM;
			SampleTaken := TRUE;
			Timer(IN := FALSE);	// Reset timer
		ELSE
			SampleTaken := FALSE;
		END_IF;

	END_IF

END_PROGRAM
```

### Program Logical/Doctoring/HS_Inp_Doct (IEC)

#### Variables.var
```iecst
VAR
	i : USINT;
	HSCounter : LCCounter;
	initialize : BOOL;
	UnwindFilt : LCPT1;
	WindFilt : LCPT1;
	Time_1sec : TON_10ms;
	Old_EncValue : INT;
	Diff_EncValue : INT;
	PulsesPerMin : UDINT;
	UnWindRPM_Scal : LCScINT;
	WindRPM_Scal : LCScINT;
	Numerator : UDINT;
	Denominator : UDINT;
	DriveCurrent_Scal : LCScINT;
	DriveRPM_Scal : LCScINT;
	DriveTorq_Scal : LCScINT;
	DriveFreq_Scal : LCScINT;
	j : USINT;
	Old_AxisMotor : INT;
END_VAR
```

#### HS_Inp_Cyclic.st
```iecst
PROGRAM _CYCLIC
	// Time base counter
	HSCounter();

	IF(initialize = 1)THEN
		// Initialize all filters

		UnwindFilt.x	:= 0;
		UnwindFilt.t		:= UnWind.RPM.Actual.Scale.Filter_tim;
		UnwindFilt.basetime	:= HSCounter.mscnt;

		WindFilt.x		:= 0;
		WindFilt();

		IF(UnWind.RPM.PulsesPerRev = 0)THEN
			UnWind.RPM.PulsesPerRev := 1;
		END_IF

		IF(Wind.RPM.PulsesPerRev= 0)THEN
			Wind.RPM.PulsesPerRev := 1;
		END_IF

		initialize := 0;

		Time_1sec.IN	:= 1;
		Old_EncValue	:= Enc_Value;

		AI1[1]	:= AI1[0];
		AI1[2]	:= AI1[1];
		AI1[3]	:= AI1[2];

	ELSE
		// CALCULATE RPM AND MPM OF IDLER AXIS

		IF(Time_1sec.Q = 1)THEN
			PulsesPerMin	:= (Enc_Value - Old_EncValue)*60;
			Time_1sec.IN	:= 0;
		ELSIF (Time_1sec.IN = 0)THEN
			Old_EncValue	:= Enc_Value;
			Time_1sec.IN	:= 1;
		END_IF

		Idler.RPM.ActRPM := UDINT_TO_INT(PulsesPerMin)/Idler.PulsesPerRev;
		Idler.MPM.ActMPM := (314 * Idler.MPM.InpDia * Idler.RPM.ActRPM)/1000; // Idler Roller MPM (in 0.01 MPM) -> which is the system MPM

		//Filter the Winder & UnWinder RPM values read from the Drive
		UnwindFilt.x		:= DINT_TO_INT(Drive_RW[0].Read_DINT[2]);
		UnwindFilt.t		:= UnWind.RPM.Actual.Scale.Filter_tim;
		UnwindFilt.basetime	:= HSCounter.mscnt;
		UnwindFilt();
		UnWind.RPM.Actual.Input_Val	:= UnwindFilt.y;

		WindFilt.x			:= DINT_TO_INT(Wind.Drive.ActRPM/10);
		WindFilt.t			:= Wind.RPM.Actual.Scale.Filter_tim;
		WindFilt.basetime	:= HSCounter.mscnt;
		WindFilt();
		Wind.RPM.Actual.Input_Val	:= WindFilt.y;

		//Calculate the RPM of Winder & Unwinder after filtering of Drive RPM & Scaling the value
		UnWindRPM_Scal.x		:= UnWind.RPM.Actual.Input_Val;
		UnWindRPM_Scal();
		UnWind.RPM.ActualRPM	:= UnWindRPM_Scal.y;

		WindRPM_Scal.x			:= Wind.RPM.Actual.Input_Val;
		WindRPM_Scal();
		Wind.RPM.ActualRPM		:= WindRPM_Scal.y;

		// CALCULATE DIAMETER OF WINDER AND UNWINDER
		IF(UnWind.RPM.ActualRPM > 0)THEN
			Numerator			:= INT_TO_UDINT(Idler.MPM.ActMPM * 1000);
			Denominator			:= INT_TO_UDINT(UnWind.RPM.ActualRPM * 314);
			UnWind.Dia.ActDia	:= UDINT_TO_INT(Numerator/Denominator) - UnWind.Dia.MinDia; // Winder DIA UNIT 0.01
		END_IF

		IF(Wind.RPM.ActualRPM > 0)THEN
			Numerator			:= INT_TO_UDINT(Idler.MPM.ActMPM * 1000);
			Denominator			:= INT_TO_UDINT(Wind.RPM.ActualRPM * 314);
			Wind.Dia.ActDia		:= UDINT_TO_INT(Numerator/Denominator) + Wind.Dia.MinDia; // Winder DIA UNIT 0.01
		END_IF

		//Just assign
		UnWind.Drive.ActFreq	:= DINT_TO_INT(Drive_RW[0].Read_UDINT[0]);
		UnWind.Drive.ActRPM		:= UnWind.Drive.ActRPM;
		UnWind.Drive.ActualAmp	:= UnWind.Drive.ActualAmp;
		UnWind.Drive.ActualTrq	:= UnWind.Drive.ActualTrq;

	END_IF

	Time_1sec();

END_PROGRAM
```

#### HS_Inp_Init.st
```iecst
PROGRAM _INIT
	(* Insert code here *)
	initialize	:= 1;

	(*Input of Tension Sensor for 4 axes except main drive *)
	AI1[0]	:= 0;	(*Unwinder Loadcell *)
	AI1[1]	:= 0;	(* Infeed Loadcell *)
	AI1[2]	:= 0;	(* Outfeed Loadcell *)
	AI1[3]	:= 0;	(* Winder Load cell *)

	AO1[0]	:= 0;
	AO1[1]	:= 0;
	AO1[2]	:= 0;
	AO1[3]	:= 0;

	DI1[0]	:= 0;
	DI1[1]	:= 0;
	DI1[2]	:= 0;
	DI1[3]	:= 0;
	DI1[4]	:= 0;
	DI1[5]	:= 0;
	DI1[6]	:= 0;
	DI1[7]	:= 0;
	DI1[8]	:= 0;
	DI1[9]	:= 0;
	DI1[10]	:= 0;
	DI1[11]	:= 0;

	DI2[0]	:= 0;
	DI2[1]	:= 0;
	DI2[2]	:= 0;
	DI2[3]	:= 0;
	DI2[4]	:= 0;
	DI2[5]	:= 0;
	DI2[6]	:= 0;
	DI2[7]	:= 0;
	DI2[8]	:= 0;
	DI2[9]	:= 0;
	DI2[10]	:= 0;
	DI2[11]	:= 0;

	DO1[0]	:= 0;
	DO1[1]	:= 0;
	DO1[2]	:= 0;
	DO1[3]	:= 0;
	DO1[4]	:= 0;
	DO1[5]	:= 0;
	DO1[6]	:= 0;
	DO1[7]	:= 0;
	DO1[8]	:= 0;
	DO1[9]	:= 0;
	DO1[10]	:= 0;
	DO1[11]	:= 0;

	DO2[0]	:= 0;
	DO2[1]	:= 0;
	DO2[2]	:= 0;
	DO2[3]	:= 0;
	DO2[4]	:= 0;
	DO2[5]	:= 0;
	DO2[6]	:= 0;
	DO2[7]	:= 0;
	DO2[8]	:= 0;
	DO2[9]	:= 0;
	DO2[10]	:= 0;
	DO2[11]	:= 0;

	FOR i := 0 TO 1 DO
		FOR j := 0 TO 9 DO
			Drive_RW[i].Write_UINT[j]	:= 0;
			Drive_RW[i].Write_DINT[j]	:= 0;
			Drive_RW[i].Read_DINT[j]	:= 0;
		END_FOR
	END_FOR

	UnWind.Drive.ActFreq		:= 0;
	UnWind.Drive.ActRPM			:= 0;
	UnWind.Drive.ActualAmp		:= 0;
	UnWind.Drive.ActualTrq		:= 0;
	UnWind.Drive.Drive_Enable	:= 0;
	UnWind.Drive.Drive_Healthy	:= 0;

	Wind.Drive.ActFreq			:= 0;
	Wind.Drive.ActRPM			:= 0;
	Wind.Drive.ActualAmp		:= 0;
	Wind.Drive.ActualTrq		:= 0;
	Wind.Drive.Drive_Enable		:= 0;
	Wind.Drive.Drive_Healthy	:= 0;

	i	:= 0;

	IF(Idler.PulsesPerRev = 0)THEN
		Idler.PulsesPerRev	:= 1;
	END_IF

	IF(UnWind.RPM.Actual.Scale.Filter_tim = 0)THEN
		UnWind.RPM.Actual.Scale.Filter_tim	:= 15;
	END_IF

	UnwindFilt.enable	:= 1;
	UnwindFilt.set		:= FALSE;
	UnwindFilt.yset		:= 0;

	IF(Wind.RPM.Actual.Scale.Filter_tim = 0)THEN
		Wind.RPM.Actual.Scale.Filter_tim	:= 15;
	END_IF

	WindFilt.enable	:= 1;
	WindFilt.set		:= FALSE;
	WindFilt.yset		:= 0;

	UnWind.Enable	:= 1;
	UnWind.MPM.Enable	:= 1;

	IF((UnWind.RPM.Actual.Scale.InMin = 0)OR(UnWind.RPM.Actual.Scale.InMax = 0))THEN
		UnWind.RPM.Actual.Scale.InMin	:= 1;
		UnWind.RPM.Actual.Scale.InMax	:= 1;
	END_IF

	IF((UnWind.RPM.Actual.Scale.OutMin = 0)OR(UnWind.RPM.Actual.Scale.OutMax = 0))THEN
		UnWind.RPM.Actual.Scale.OutMin	:= 1;
		UnWind.RPM.Actual.Scale.OutMax	:= 1;
	END_IF

	IF((Wind.RPM.Actual.Scale.InMin = 0)OR(Wind.RPM.Actual.Scale.InMax = 0))THEN
		Wind.RPM.Actual.Scale.InMin	:= 1;
		Wind.RPM.Actual.Scale.InMax	:= 1;
	END_IF

	IF((Wind.RPM.Actual.Scale.OutMin = 0)OR(Wind.RPM.Actual.Scale.OutMax = 0))THEN
		Wind.RPM.Actual.Scale.OutMin	:= 1;
		Wind.RPM.Actual.Scale.OutMax	:= 1;
	END_IF

	UnWindRPM_Scal.x1	:= UnWind.RPM.Actual.Scale.InMin;
	UnWindRPM_Scal.x2	:= UnWind.RPM.Actual.Scale.InMax;
	UnWindRPM_Scal.y1	:= UnWind.RPM.Actual.Scale.OutMin;
	UnWindRPM_Scal.y2	:= UnWind.RPM.Actual.Scale.OutMax;

	WindRPM_Scal.x1		:= Wind.RPM.Actual.Scale.InMin;
	WindRPM_Scal.x2		:= Wind.RPM.Actual.Scale.InMax;
	WindRPM_Scal.y1		:= Wind.RPM.Actual.Scale.OutMin;
	WindRPM_Scal.y2		:= Wind.RPM.Actual.Scale.OutMax;

	(* Scaling drive parameters *)
	(* TORQUE *)
	IF((UnWind.Drive.Trq_Scal.InMin = 0)OR(UnWind.Drive.Trq_Scal.InMax = 0))THEN
		UnWind.Drive.Trq_Scal.InMin	:= 1;
		UnWind.Drive.Trq_Scal.InMax	:= 1;
	END_IF

	IF((UnWind.Drive.Trq_Scal.OutMin = 0)OR(UnWind.Drive.Trq_Scal.OutMax = 0))THEN
		UnWind.Drive.Trq_Scal.OutMin 	:= 1;
		UnWind.Drive.Trq_Scal.OutMax := 1;
	END_IF

	IF((Wind.Drive.Trq_Scal.InMin = 0)OR(Wind.Drive.Trq_Scal.InMax = 0))THEN
		Wind.Drive.Trq_Scal.InMin	:= 1;
		Wind.Drive.Trq_Scal.InMax	:= 1;
	END_IF

	IF((Wind.Drive.Trq_Scal.OutMin = 0)OR(Wind.Drive.Trq_Scal.OutMax = 0))THEN
		Wind.Drive.Trq_Scal.OutMin 	:= 1;
		Wind.Drive.Trq_Scal.OutMax := 1;
	END_IF

	(* CURRENT *)
	IF((UnWind.Drive.Current_Scal.InMin = 0)OR(UnWind.Drive.Current_Scal.InMax = 0))THEN
		UnWind.Drive.Current_Scal.InMin	:= 1;
		UnWind.Drive.Current_Scal.InMax	:= 1;
	END_IF

	IF((UnWind.Drive.Current_Scal.OutMin = 0)OR(UnWind.Drive.Current_Scal.OutMax = 0))THEN
		UnWind.Drive.Current_Scal.OutMin 	:= 1;
		UnWind.Drive.Current_Scal.OutMax := 1;
	END_IF

	IF((Wind.Drive.Current_Scal.InMin = 0)OR(Wind.Drive.Current_Scal.InMax = 0))THEN
		Wind.Drive.Current_Scal.InMin	:= 1;
		Wind.Drive.Current_Scal.InMax	:= 1;
	END_IF

	IF((Wind.Drive.Current_Scal.OutMin = 0)OR(Wind.Drive.Current_Scal.OutMax = 0))THEN
		Wind.Drive.Current_Scal.OutMin 	:= 1;
		Wind.Drive.Current_Scal.OutMax := 1;
	END_IF

	(* RPM *)
	IF((UnWind.Drive.RPM_Scal.InMin = 0)OR(UnWind.Drive.RPM_Scal.InMax = 0))THEN
		UnWind.Drive.RPM_Scal.InMin		:= 1;
		UnWind.Drive.RPM_Scal.InMax		:= 1;
	END_IF

	IF((UnWind.Drive.RPM_Scal.OutMin = 0)OR(UnWind.Drive.RPM_Scal.OutMax = 0))THEN
		UnWind.Drive.RPM_Scal.OutMin	:= 1;
		UnWind.Drive.RPM_Scal.OutMax	:= 1;
	END_IF

	IF((Wind.Drive.RPM_Scal.InMin = 0)OR(Wind.Drive.RPM_Scal.InMax = 0))THEN
		Wind.Drive.RPM_Scal.InMin	:= 1;
		Wind.Drive.RPM_Scal.InMax	:= 1;
	END_IF

	(* FREQUENCY *)
	IF((UnWind.Drive.Freq_Scal.InMin = 0)OR(UnWind.Drive.Freq_Scal.InMax = 0))THEN
		UnWind.Drive.Freq_Scal.InMin	:= 1;
		UnWind.Drive.Freq_Scal.InMax	:= 1;
	END_IF

	IF((UnWind.Drive.Freq_Scal.OutMin = 0)OR(UnWind.Drive.Freq_Scal.OutMax = 0))THEN
		UnWind.Drive.Freq_Scal.OutMin 	:= 1;
		UnWind.Drive.Freq_Scal.OutMax := 1;
	END_IF

	IF((Wind.Drive.Freq_Scal.InMin = 0)OR(Wind.Drive.Freq_Scal.InMax = 0))THEN
		Wind.Drive.Freq_Scal.InMin	:= 1;
		Wind.Drive.Freq_Scal.InMax	:= 1;
	END_IF

	IF((Wind.Drive.Freq_Scal.OutMin = 0)OR(Wind.Drive.Freq_Scal.OutMax = 0))THEN
		Wind.Drive.Freq_Scal.OutMin	:= 1;
		Wind.Drive.Freq_Scal.OutMax := 1;
	END_IF

	Time_1sec.PT	:= 100;

END_PROGRAM
```

### Program Logical/Doctoring/LS_Inp_OP (IEC)

#### Cyclic.st
```iecst
PROGRAM _CYCLIC
	(* Insert code here *)
	DigInp.Emergency_OK		:= DI1[0];
	DigInp.Jog_mode			:= DI1[1];
	Mode_Intermediate		:= DI1[2];
	DigInp.MPM_Increase		:= DI1[3];
	DigInp.MPM_Decrease		:= DI1[4];
	DigInp.Safety_Trip		:= DI1[5];

	IF(check_init = 1)THEN
		IF (Mode_Intermediate = 1)THEN
			Alarm_mc[0]	:= 1;
			mode_allow	:= 0;
		ELSE
			mode_allow	:= 1;
		END_IF
		check_init	:= 0;
	END_IF

	IF(mode_allow = 1)THEN
		IF((DigInp.Jog_mode = 0)AND(Mode_Intermediate = 1))THEN
			DigInp.Production_mode	:= Mode_Intermediate;
		ELSE
			DigInp.Production_mode	:= 0;
		END_IF
	ELSE
		DigInp.Production_mode	:= 0;
	END_IF

	IF(DigInp.Production_mode = 1)THEN
		IF(DigInp.MPM_Increase = 1)THEN
			MPMIncTime.IN	:= 1;
			IF(MPMIncTime.ET < 500)THEN
				inc_cnt	:= inc_cnt + 1;
				IF(inc_cnt >= 50)THEN
					UnWind.MPM.SetMPM	:= UnWind.MPM.SetMPM + 1;
					inc_cnt	:= 0;
				END_IF
			ELSIF(MPMIncTime.ET < 800)THEN
				inc_cnt	:= inc_cnt + 1;
				IF(inc_cnt >= 50)THEN
					UnWind.MPM.SetMPM	:= UnWind.MPM.SetMPM + 10;
					inc_cnt	:= 0;
				END_IF
			ELSIF(MPMIncTime.ET < 1000)THEN
				inc_cnt	:= inc_cnt + 1;
				IF(inc_cnt >= 50)THEN
					UnWind.MPM.SetMPM	:= UnWind.MPM.SetMPM + 100;
					inc_cnt	:= 0;
				END_IF
			END_IF
		ELSE
			MPMIncTime.IN	:= 0;
			inc_cnt			:= 0;
		END_IF

		IF(DigInp.MPM_Decrease = 1)THEN
			MPMDecTime.IN	:= 1;
			IF(MPMDecTime.ET < 500)THEN
				dec_cnt	:= dec_cnt + 1;
				IF(dec_cnt >= 50)THEN
					UnWind.MPM.SetMPM	:= UnWind.MPM.SetMPM - 1;
					dec_cnt	:= 0;
				END_IF
			ELSIF(MPMDecTime.ET < 800)THEN
				dec_cnt	:= dec_cnt + 1;
				IF(dec_cnt >= 50)THEN
					UnWind.MPM.SetMPM	:= UnWind.MPM.SetMPM - 10;
					dec_cnt	:= 0;
				END_IF
			ELSIF(MPMDecTime.ET < 1000)THEN
				dec_cnt	:= dec_cnt + 1;
				IF(dec_cnt >= 50)THEN
					UnWind.MPM.SetMPM	:= UnWind.MPM.SetMPM - 100;
					dec_cnt	:= 0;
				END_IF
			END_IF
		ELSE
			MPMDecTime.IN	:= 0;
			dec_cnt			:= 0;
		END_IF
	ELSE
		MPMDecTime.IN	:= 0;
		dec_cnt			:= 0;
		MPMIncTime.IN	:= 0;
		inc_cnt			:= 0;
	END_IF

	IF(DigInp.Production_mode = 1)THEN
		Drive_RW[0].Write_DINT[0]	:= INT_TO_DINT(UnWind.MPM.SetMPM);
		Drive_RW[1].Write_DINT[0]	:= INT_TO_DINT(UnWind.RPM.Actual.Input_Val);
	ELSIF(DigInp.Jog_mode = 1)THEN
		Drive_RW[0].Write_DINT[0]	:= INT_TO_DINT(UnWind.MPM.SetMPM);
		Drive_RW[1].Write_DINT[0]	:= INT_TO_DINT(Wind.MPM.SetMPM);
//		Drive_RW[0].Write_UINT[0]	:= UnWind.MPM.SetMPM;
//		Drive_RW[1].Write_UINT[0]	:= Wind.MPM.SetMPM;
	ELSE
		Drive_RW[0].Write_UINT[0]	:= 0;
		Drive_RW[1].Write_UINT[0]	:= 0;
		UnWind.MPM.SetMPM			:= 0;
		Wind.MPM.SetMPM				:= 0;
	END_IF

	MPMIncTime();
	MPMDecTime();

	(* Configure the Outputs from here *)

	IF ((UnWind.Drive.Drive_Healthy	= 1)AND(Wind.Drive.Drive_Healthy = 1))THEN
		DO1[0]	:= 1;
		DO1[1]	:= 1;
	ELSE
		DO1[0]	:= 0;
		DO1[1]	:= 0;
	END_IF

END_PROGRAM
```

#### Init.st
```iecst
PROGRAM _INIT
	(* Insert code here *)
	memset(ADR(DigInp), 0, SIZEOF(DigInp));
	MPMIncTime.IN	:= 0;
	MPMIncTime.PT	:= 9999;

	MPMDecTime.IN	:= 0;
	MPMDecTime.PT	:= 9999;

	check_init	:= 1;

END_PROGRAM
```

### Program Logical/Doctoring/Simulate (IEC)

#### Variables.var
```iecst
VAR
	cnt : INT;
	x : INT;
	var : INT;
END_VAR
```

#### Cyclic.st
```iecst
PROGRAM _CYCLIC
	(* Insert code here *)
	cnt	:= cnt + 1;
	x	:= cnt MOD 3;

	IF(cnt < 50) THEN
		IF(x = 0)THEN
			var	:= var + 5;
		ELSIF (x = 1)THEN
			var	:= var - 2;
		ELSE
			var	:= var - 1;
		END_IF
	ELSIF (cnt < 100)THEN
		IF(x = 0)THEN
			var	:= var + 5;
		ELSIF (x = 1)THEN
			var	:= var - 2;
		ELSE
			var	:= var - 1;
		END_IF
	END_IF

	IF(cnt >= 100)THEN
		cnt	:= 0;
		var	:= 500;
	END_IF

	Drive_RW[0].Read_DINT[2]	:= var;

END_PROGRAM
```

#### Init.st
```iecst
PROGRAM _INIT
	(* Insert code here *)
	var	:= 500;
	cnt	:= 0;
END_PROGRAM
```

- Visualisation Logical/Vis (not shown)

### Program Logical/Alarms (IEC)

#### Cyclic.st
```iecst
PROGRAM _CYCLIC
	(* Insert code here *)
	Alarm_cnt	:= 0;

	FOR i := 0 TO 99 DO
		IF(Alarm_mc[i] > 0)THEN
			Alarm_cnt	:= Alarm_cnt + 1;
		END_IF
	END_FOR

	IF(Alarm_cnt > 0)THEN
		Statusdp_blink	:= 1;
		IF(count = 0)THEN
			Blink_ON.IN	:= 1;
			IF(Blink_ON.Q = 1)THEN
				count := 1;
				Blink_ON.IN	:= 0;
			END_IF
		ELSE
			Blink_OFF.IN	:= 1;
			IF(Blink_OFF.Q = 1)THEN
				count := 0;
				Blink_OFF.IN := 0;
			END_IF
		END_IF

	ELSE
		Blink_ON.IN		:= 0;
		Blink_OFF.IN	:= 0;
		Statusdp_blink	:= 0;
	END_IF

	Blink_ON(IN := TRUE, PT := 1);	//1 × 10ms = 10 milliseconds
	Blink_OFF(IN := TRUE, PT := 1);

END_PROGRAM
```

#### Init.st
```iecst
PROGRAM _INIT
	(* Insert code here *)
	Statusdp_alarm	:= 0;
	Alarm_cnt		:= 0;
	Alarm_new		:= 0;
	Blink_ON.IN		:= 0;
	Blink_ON.PT		:= 100;
	Blink_OFF.IN	:= 0;
	Blink_OFF.PT	:= 100;

	memset(ADR(Alarm_mc), 0, SIZEOF(Alarm_mc));

END_PROGRAM
```

### Program Logical/Mot_Tun

#### Cyclic.st
```iecst
PROGRAM _CYCLIC
	(* Insert code here *)
	IF ( Save = 1 ) THEN
		CASE Axis_Motor OF
			0: 		// None

			1:		// Unwinder
				UnWind.MotorRating.RatedFreq 	:= TempFreq;
				UnWind.MotorRating.RatedCurrent := TempCurrent;
				UnWind.MotorRating.RatedVoltage := TempVoltage;
				UnWind.MotorRating.RatedSpeed	:= TempSpeed;
				UnWind.MotorRating.RatedPF 		:= TempPF;
				CopytoDrv						:= 1;
				plc_node						:= 3;

			2:		// Winder
				Wind.MotorRating.RatedFreq 		:= TempFreq;
				Wind.MotorRating.RatedCurrent 	:= TempCurrent;
				Wind.MotorRating.RatedVoltage 	:= TempVoltage;
				Wind.MotorRating.RatedSpeed		:= TempSpeed;
				Wind.MotorRating.RatedPF 		:= TempPF;
				CopytoDrv						:= 1;
				plc_node						:= 4;

			3:		// Infeed

			4:		// Outfeed

			5:		// Main

		END_CASE
		Save		:= 0;
		Axis_Motor	:= 0;
		Old_AxisMotor	:= Axis_Motor;
	ELSE
		IF(Axis_Motor <> Old_AxisMotor)THEN
			CASE Axis_Motor OF
				0: 		// None
					TempFreq	:= 0;
					TempCurrent	:= 0;
					TempVoltage	:= 0;
					TempSpeed	:= 0;
					TempPF		:= 0;

				1:		// Unwinder
					TempFreq	:= UnWind.MotorRating.RatedFreq;
					TempCurrent	:= UnWind.MotorRating.RatedCurrent;
					TempVoltage	:= UnWind.MotorRating.RatedVoltage;
					TempSpeed	:= UnWind.MotorRating.RatedSpeed;
					TempPF		:= UnWind.MotorRating.RatedPF;

				2:		// Winder
					TempFreq	:= Wind.MotorRating.RatedFreq;
					TempCurrent	:= Wind.MotorRating.RatedCurrent;
					TempVoltage	:= Wind.MotorRating.RatedVoltage;
					TempSpeed	:= Wind.MotorRating.RatedSpeed;
					TempPF		:= Wind.MotorRating.RatedPF;

				3:		// Infeed
					TempFreq	:= 0;
					TempCurrent	:= 0;
					TempVoltage	:= 0;
					TempSpeed	:= 0;
					TempPF		:= 0;

				4:		// Outfeed
					TempFreq	:= 0;
					TempCurrent	:= 0;
					TempVoltage	:= 0;
					TempSpeed	:= 0;
					TempPF		:= 0;

				5:		// Main
					TempFreq	:= 0;
					TempCurrent	:= 0;
					TempVoltage	:= 0;
					TempSpeed	:= 0;
					TempPF		:= 0;

			END_CASE
			Old_AxisMotor	:= Axis_Motor;
		END_IF
	END_IF

	CASE motordata_step OF
		0:
			IF(CopytoDrv = 1)THEN
				motordata_step	:= 1;
				dlycnt1			:= 0;
			END_IF

		1:
			SDOWrite.node		:= plc_node;
			SDOWrite.pData		:= ADR(TempFreq);
			SDOWrite.datalen 	:= 4; //Data length, 2 bytes for 16-bit parameter
			SDOWrite.index 		:= 16#2005;
			SDOWrite.subindex	:= 6;
			SDOWrite.enable		:= 1;
			dlycnt1				:= dlycnt1 + 1;
			IF(dlycnt1 > 1)THEN
				IF (SDOWrite.status = 0) THEN
					SDOWrite.enable	:= 0;
					motordata_step	:= 2;
					dlycnt1			:= 0;
				ELSIF(SDOWrite.status <> 65535)THEN
					SDOWrite.enable	:= 0;
					motordata_step	:= 0;
					CopytoDrv		:= 0;
				END_IF
			END_IF

		2:
			// Write Motor Current
			SDOWrite.node		:= plc_node;
			SDOWrite.pData		:= ADR(TempCurrent);
			SDOWrite.datalen 	:= 4; //Data length, 2 bytes for 16-bit parameter
			SDOWrite.index 		:= 16#2005;
			SDOWrite.subindex	:= 7;
			SDOWrite.enable		:= 1;
			dlycnt1				:= dlycnt1 + 1;
			IF(dlycnt1 > 1)THEN
				IF (SDOWrite.status = 0) THEN
					SDOWrite.enable	:= 0;
					motordata_step	:= 3;
					dlycnt1			:= 0;
				ELSIF(SDOWrite.status <> 65535)THEN
					SDOWrite.enable	:= 0;
					motordata_step	:= 0;
					CopytoDrv		:= 0;
				END_IF
			END_IF

		3:
			SDOWrite.node		:= plc_node;
			SDOWrite.pData		:= ADR(TempVoltage);
			SDOWrite.datalen 	:= 2; //Data length, 2 bytes for 16-bit parameter
			SDOWrite.index 		:= 16#2005; //Index = 0x2000 + Menu Number
			SDOWrite.subindex	:= 9;
			SDOWrite.enable		:= 1;
			dlycnt1				:= dlycnt1 + 1;
			IF(dlycnt1 > 1)THEN
				IF (SDOWrite.status = 0) THEN
					SDOWrite.enable	:= 0;
					motordata_step	:= 4;
					dlycnt1			:= 0;
				ELSIF(SDOWrite.status <> 65535)THEN
					SDOWrite.enable	:= 0;
					motordata_step	:= 0;
					CopytoDrv		:= 0;
				END_IF
			END_IF

		4:
			SDOWrite.node		:= plc_node;
			SDOWrite.pData		:= ADR(TempSpeed);
			SDOWrite.datalen 	:= 4; //Data length, 2 bytes for 16-bit parameter
			SDOWrite.index 		:= 16#2005; //Index = 0x2000 + Menu Number
			SDOWrite.subindex	:= 8;
			SDOWrite.enable		:= 1;
			dlycnt1				:= dlycnt1 + 1;
			IF(dlycnt1 > 1)THEN
				IF (SDOWrite.status = 0) THEN
					SDOWrite.enable	:= 0;
					motordata_step	:= 5;
					dlycnt1			:= 0;
				ELSIF(SDOWrite.status <> 65535)THEN
					SDOWrite.enable	:= 0;
					motordata_step	:= 0;
					CopytoDrv		:= 0;
				END_IF
			END_IF
		5:
			SDOWrite.node		:= plc_node;
			SDOWrite.pData		:= ADR(TempPF);
			SDOWrite.datalen 	:= 2; //Data length, 2 bytes for 16-bit parameter
			SDOWrite.index 		:= 16#2005; //Index = 0x2000 + Menu Number
			SDOWrite.subindex	:= 10;
			SDOWrite.enable		:= 1;
			dlycnt1				:= dlycnt1 + 1;
			IF(dlycnt1 > 1)THEN
				IF (SDOWrite.status = 0) THEN
					SDOWrite.enable	:= 0;
					motordata_step	:= 0;
					dlycnt1			:= 0;
					CopytoDrv		:= 0;
				ELSIF(SDOWrite.status <> 65535)THEN
					SDOWrite.enable	:= 0;
					motordata_step	:= 0;
					CopytoDrv		:= 0;
				END_IF
			END_IF
	END_CASE

	IF(Tune_Enable = 1)THEN
		Old_AxisMotorTune	:= Axis_MotorTune;
	END_IF

	(* Initial Power Up Configuring the Control Word to Read Freq. Command from Preset-1 & disable other preset values
	& enable the Control *)

	CASE wr_step OF
		0:
			IF(Tune_Enable = 1)THEN
				IF(Axis_MotorTune = 1)THEN
					plc_node	:= 3;
				ELSIF(Axis_MotorTune = 2)THEN
					plc_node	:= 4;
				END_IF
				wr_step		:= 1; //Tune UnWinder motor
				dlycnt	:= 0;
			END_IF

		1:
			//Disable the Control Enable
			Control_Enable		:= 0;

			SDOTune_wr.node		:= plc_node;
			SDOTune_wr.pData	:= ADR(Control_Enable);
			SDOTune_wr.datalen 	:= 1; //Data length, 2 bytes for 16-bit parameter
			SDOTune_wr.index 	:= 16#2006;
			SDOTune_wr.subindex	:= 43;
			SDOTune_wr.enable	:= 1;
			dlycnt				:= dlycnt + 1;
			IF(dlycnt > 1)THEN
				IF (SDOTune_wr.status = 0) THEN
					SDOTune_wr.enable	:= 0;
					wr_step				:= 2;
					dlycnt				:= 0;
				ELSIF(SDOTune_wr.status <> 65535)THEN
					SDOTune_wr.enable	:= 0;
				END_IF
			END_IF
		2:
			//Confirm that the Drive is not Active

			SDOTune_rd.node		:= plc_node;
			SDOTune_rd.pData 	:= ADR(Status_WORD); //Data to be read into here
			SDOTune_rd.datalen	:= 2; //Data length, 2 bytes for 16-bit parameter
			SDOTune_rd.index 	:= 16#200A;
			SDOTune_rd.subindex	:= 40;
			SDOTune_rd.enable	:= 1;
			dlycnt				:= dlycnt + 1;
			IF(dlycnt > 1)THEN
				IF (SDOTune_rd.status = 0) THEN
					SDOTune_rd.enable	:= 0;
					dlycnt				:= 0;
					IF(Status_WORD.1 = 0)THEN
						wr_step			:= 3;
					END_IF
				ELSIF(SDOTune_rd.status <> 65535)THEN
					SDOTune_rd.enable	:= 0;
				END_IF
			END_IF

		3:
			// Set the Auto Tune Bit
			Tune_Start			:= 2;

			SDOTune_wr.pData	:= ADR(Tune_Start);
			SDOTune_wr.datalen 	:= 1; //Data length, 2 bytes for 16-bit parameter
			SDOTune_wr.index 	:= 16#2005;
			SDOTune_wr.subindex	:= 12;
			SDOTune_wr.enable	:= 1;
			dlycnt				:= dlycnt + 1;
			IF(dlycnt > 3)THEN
				IF (SDOTune_wr.status = 0) THEN
					SDOTune_wr.enable	:= 0;
					wr_step			:= 4;
					dlycnt			:= 0;
					firstchck		:= 1;
				ELSIF(SDOTune_wr.status <> 65535)THEN
					SDOTune_wr.enable	:= 0;
				END_IF
			END_IF
		4:
			//Disable the Control Enable
			Control_Enable		:= 1;

			SDOTune_wr.node		:= plc_node;
			SDOTune_wr.pData	:= ADR(Control_Enable);
			SDOTune_wr.datalen 	:= 1; //Data length, 2 bytes for 16-bit parameter
			SDOTune_wr.index 	:= 16#2006;
			SDOTune_wr.subindex	:= 43;
			SDOTune_wr.enable	:= 1;
			dlycnt				:= dlycnt + 1;
			IF(dlycnt > 1)THEN
				IF (SDOTune_wr.status = 0) THEN
					SDOTune_wr.enable	:= 0;
					wr_step				:= 5;
					dlycnt				:= 0;
				ELSIF(SDOTune_wr.status <> 65535)THEN
					SDOTune_wr.enable	:= 0;
				END_IF
			END_IF

		5:
			// Check if Auto Tune is complete
			SDOTune_rd.node		:= plc_node;
			SDOTune_rd.pData 	:= ADR(Status_WORD);
			SDOTune_rd.datalen	:= 1;
			SDOTune_rd.index 	:= 16#2005;
			SDOTune_rd.subindex	:= 12;

			IF(firstchck = 1)THEN
				SDOTune_rd.enable	:= 1;
			ELSIF(chkdly > 50)THEN
				SDOTune_rd.enable	:= 1;
				chkdly				:= 0;
			END_IF

			dlycnt			:= dlycnt + 1;

			IF(dlycnt > 1)THEN
				IF (SDOTune_rd.status = 0) THEN
					SDOTune_rd.enable	:= 0;
					IF(Status_WORD = 0)THEN
						wr_step		:= 0;
						Tune_Enable	:= 0;
						dlycnt		:= 0;
						chkdly		:= 0;
					END_IF
				ELSIF(SDOTune_rd.status <> 65535)THEN
					SDOTune_rd.enable	:= 0;
				END_IF
			END_IF

			IF(Status_WORD = 2)THEN
				chkdly	:= chkdly + 1;
			END_IF

	END_CASE

	SDOTune_wr();
	SDOTune_rd();
	SDOWrite();

END_PROGRAM
```

#### Init.st
```iecst
PROGRAM _INIT
	(* Insert code here *)
	TempFreq	:= 0;
	TempCurrent	:= 0;
	TempVoltage	:= 0;
	TempSpeed	:= 0;
	TempPF		:= 0;

	Save			:= 1;
	Axis_Motor		:= 0;
	Old_AxisMotor	:= 0;

	SDOTune_rd.enable	:= 0;
	SDOTune_rd.pDevice 	:= ADR(PLC_INTF); //POWERLINK interface on MN (PLC) ‘IF1’
	SDOTune_rd.node 	:= plc_node; //Node address is set to 3

	SDOTune_wr.enable	:= 0;
	SDOTune_wr.pDevice	:= ADR(PLC_INTF);
	SDOTune_wr.node		:= plc_node;

END_PROGRAM
```
